METHOD SetPowerMode : BOOL
VAR_INST
	WriteReg	:	FB_MBWriteSingleReg;
	Value 		:	WORD 	:= 1;
	StartWrite	:	BOOL	:= FALSE;
	bCommBusy	:	BOOL;
	bComError	:	BOOL;
	errID		:	UDINT;
	TransmissionDone 	: 	f_trig;
	ComTrigger	:	Ton := (PT := TIME#200MS);
	ComRetryCounter	:	USINT	:= 0;
END_VAR	

VAR

END_VAR

Value := ePowerControl.Stay; //default command is: Do nothing
//it may also work if we just keep sending "poweron" if b_HVDC_Required is true. But this doesn't seem to be the way they intended.

IF Set.b_HVDC_Required AND (BMSGet.BattInfo.ui_BMS_PowerOnStatus = ePowerOnStatus.Off) THEN	//send poweron if system not already on
	Value := ePowerControl.PowerOn;
ELSIF (NOT Set.b_HVDC_Required) AND (BMSGet.BattInfo.ui_BMS_PowerOnStatus = ePowerOnStatus.On) THEN //send poweroff if system not already off
	Value := ePowerControl.PowerOff;
END_IF

//Write this register every second, regardless of change.
ComTrigger(in := NOT(ComTrigger.Q));

//IF BMSGet.BattInfo.ui_BMS_Status < 5 THEN
WriteReg(
	sIPAddr := Config.IP_BMS,
	nTCPPort := Config.MBPort_BMS,
	nUnitID := 255,//16#FF;
	nMBAddr := 897,
	nValue := Value,
	tTimeout := T#0S100MS,
	bExecute := ComTrigger.Q,
	bBusy => bCommBusy,
	bError => bComError,
	nErrId => errID,
);
//ELSE
//	SetPowerMode := TRUE;
//END_IF

	
TransmissionDone(CLK := bCommBusy);
	
//return true if tranmission succeeds
IF TransmissionDone.Q THEN
	IF NOT bComError THEN
		SetPowerMode := TRUE;
		ComRetryCounter := 0;
	ELSE
		COMretryCounter := COMretryCounter +1;
		IF COMRetryCounter > 5 THEN
			b_MBComErrorActive := TRUE;
		END_IF
	END_IF
END_IF
END_METHOD

ACTION SFCTipReset:
SFCTip := FALSE;
END_ACTION

END_FUNCTION_BLOCK

// ---- POUs/Objects/BMS/FB_BMS_IO.TcPOU
FUNCTION_BLOCK FB_BMS_IO

VAR_INPUT
	HWControl			:	st_BMS_IO;
END_VAR

VAR_OUTPUT
	BMSPowerControl			AT %Q* : st_BMS_IO;
END_VAR

VAR
	PowerUpDelay	:	TON := (PT := TIME#1s0ms);
END_VAR


BMSPowerControl.b_BMS_230V_Enable := HWControl.b_BMS_230V_Enable;
BMSPowerControl.b_BMS_24V_Enable	:= HWControl.b_BMS_24V_Enable;

END_FUNCTION_BLOCK

// ---- POUs/Objects/CoolingSystem/CoolingStack/FB_Heatpump.TcPOU
FUNCTION_BLOCK FB_Heatpump
VAR
	u_counter: UINT;
	InitSFC			:	FB_HeatPumpInit;
	OperationSFC	:	FB_HeatPumpOperation;
	
	//only written once at init.
	HeatPumpID		:	BYTE := 0;
END_VAR

VAR_STAT
	ui_Instancecounter : byte := 0;
END_VAR

VAR	
	MBMaster				: 	ModbusRtuMasterV2_KL6x22B;
	
	DataBuffer				:	ARRAY[0..50] OF WORD;
//	b_MBBusy				:	BOOL;
//	b_MBerr					:	BOOL;
//	ui_cbRead				:	UINT;
//	b_EnableTransmission	:	BOOL;
//	ModbusStartTrigger		:	R_Trig;
//	MBRetryCount			:	BYTE;
	
	
//	SendValue		:	WORD;
	
	OperatingPoint	:	st_OperatingPoint;
END_VAR

VAR_OUTPUT
	get			:	st_HeatpumpGet;
	MBCommBusy	:	BOOL := FALSE;
END_VAR

VAR_INPUT
	ACPowerStatus	:	BOOL;
	MBFree			:	BOOL;
END_VAR

//HeatpumpId is set once during first call
//var Stat InstanceCounter is shared between all functionblocks
IF HeatPumpId = 0 THEN
	ui_Instancecounter := ui_Instancecounter + 1;
	HeatPumpID := ui_Instancecounter ;
ELSE
	IF NOT ACPowerStatus THEN
		//Dont read all sensor data. Just monitor errors. We are not going to do anyting with the data anyway.
		InitSFC.SFCInit := TRUE;
		OperationSFC.SFCInit := TRUE;
		//OperationalSFC();
	ELSE
		InitSFC.SFCInit := FALSE;
		OperationSFC.SFCInit := FALSE;
	END_IF
END_IF

InitSFC(MBMaster := MBMaster, Get := Get, ACPowerSTatus := ACPowerStatus, HeatPumpID:=HeatPumpID);
OperationSFC(MBMaster := MBMaster, Get := Get, ACPowerSTatus := ACPowerStatus, HeatPumpID:=HeatPumpID,MBFree:=MBFree, OperatingPoint:=OperatingPoint, MBCommBusy=>MBCommbusy);

METHOD EMStop : BOOL
VAR_INPUT
END_VAR

get.HeatPumpState := eHeatpumpState.OFF;

EMstop := True;
END_METHOD

METHOD GetDiagnostics 
VAR_IN_OUT
	AddError		: ARRAY [*] OF FB_AddErrorST;
	a_ActiveEvents	: ARRAY [*] OF ST_ErrorStruct;
	w_Index			: WORD;
END_VAR

VAR_OUTPUT
	b_errorActive	: BOOL;
	b_warningActive	: BOOL;
END_VAR

VAR
	by_errCt	: BYTE;
	by_warnCt	: BYTE;
	w_ID		: WORD;
END_VAR
	(*Modbus comm fault*)	AddError[w_Index](
			in_b_ErrorTrig			:= Get.Events.b_CommError,
			out_ST_Error			:= a_ActiveEvents[w_Index],
			w_ID					:= 1 + w_ID,
			s_Message				:= 'Modbus communication error',
			e_sev					:= eSeverity.NormalShutdown,	
			in_b_AutoClear			:= FALSE,
			//in_e_ErrAckAccess		:= TRUE,
			);
		IF AddError[w_Index].b_out THEN by_errCt := by_errCt + 1; END_IF;
		w_Index := w_Index +1;
		
	(*Heatpump Compressor fault*)	AddError[w_Index](
			in_b_ErrorTrig			:= Get.Events.b_CompressorError,
			out_ST_Error			:= a_ActiveEvents[w_Index],
			w_ID					:= 2 + w_ID,
			s_Message				:= 'Heatpump Compressor fault',
			e_sev					:= eSeverity.NormalShutdown,	
			in_b_AutoClear			:= FALSE,
			//in_e_ErrAckAccess		:= TRUE,
			);
		IF AddError[w_Index].b_out THEN by_errCt := by_errCt + 1; END_IF;
		w_Index := w_Index +1;
	
	(*Heatpump Fan fault*)			AddError[w_Index](
			in_b_ErrorTrig			:= Get.Events.b_FanError,
			out_ST_Error			:= a_ActiveEvents[w_Index],
			w_ID					:= 3 + w_ID,
			s_Message				:= 'Heatpump Fan fault',
			e_sev					:= eSeverity.NormalShutdown,	
			in_b_AutoClear			:= FALSE,
			//in_e_ErrAckAccess		:= TRUE,
			);
		IF AddError[w_Index].b_out THEN by_errCt := by_errCt + 1; END_IF;
		w_Index := w_Index +1;
		
	(*HHeatpump Internal IO fault*)		AddError[w_Index](
			in_b_ErrorTrig			:= Get.Events.b_IOError ,
			out_ST_Error			:= a_ActiveEvents[w_Index],
			w_ID					:= 4 + w_ID,
			s_Message				:= 'Heatpump Internal IO fault',
			e_sev					:= eSeverity.NormalShutdown,	
			in_b_AutoClear			:= FALSE,
			//in_e_ErrAckAccess		:= TRUE,
			);
		IF AddError[w_Index].b_out THEN by_errCt := by_errCt + 1; END_IF;
		w_Index := w_Index +1;
		
	(*Heatpump pressure fault*)		AddError[w_Index](
			in_b_ErrorTrig			:= Get.Events.b_PressureError,
			out_ST_Error			:= a_ActiveEvents[w_Index],
			w_ID					:= 5 + w_ID,
			s_Message				:= 'Heatpump pressure fault',
			e_sev					:= eSeverity.NormalShutdown,	
			in_b_AutoClear			:= FALSE,
			//in_e_ErrAckAccess		:= TRUE,
			);
		IF AddError[w_Index].b_out THEN by_errCt := by_errCt + 1; END_IF;
		w_Index := w_Index +1;
		
	(*Heatpump Probe fault*)		AddError[w_Index](
			in_b_ErrorTrig			:= Get.Events.b_ProbeError,
			out_ST_Error			:= a_ActiveEvents[w_Index],
			w_ID					:= 6 + w_ID,
			s_Message				:= 'Heatpump Probe fault',
			e_sev					:= eSeverity.NormalShutdown,	
			in_b_AutoClear			:= FALSE,
			//in_e_ErrAckAccess		:= TRUE,
			);
		IF AddError[w_Index].b_out THEN by_errCt := by_errCt + 1; END_IF;
		w_Index := w_Index +1;	

	(*Heatpump Pump fault*)			AddError[w_Index](
			in_b_ErrorTrig			:= Get.Events.b_PumpError,
			out_ST_Error			:= a_ActiveEvents[w_Index],
			w_ID					:= 7 + w_ID,
			s_Message				:= 'Heatpump Pump fault',
			e_sev					:= eSeverity.NormalShutdown,	
			in_b_AutoClear			:= FALSE,
			//in_e_ErrAckAccess		:= TRUE,
			);
		IF AddError[w_Index].b_out THEN by_errCt := by_errCt + 1; END_IF;
		w_Index := w_Index +1;	

	(*Heatpump valve fault*)			AddError[w_Index](
			in_b_ErrorTrig			:= Get.Events.b_ValveError,
			out_ST_Error			:= a_ActiveEvents[w_Index],
			w_ID					:= 8 + w_ID,
			s_Message				:= 'Heatpump Valve fault',
			e_sev					:= eSeverity.NormalShutdown,	
			in_b_AutoClear			:= FALSE,
			//in_e_ErrAckAccess		:= TRUE,
			);
		IF AddError[w_Index].b_out THEN by_errCt := by_errCt + 1; END_IF;
		w_Index := w_Index +1;	

	(*Heatpump Water temperature error*)			AddError[w_Index](
			in_b_ErrorTrig			:= Get.Events.b_WaterTempError,
			out_ST_Error			:= a_ActiveEvents[w_Index],
			w_ID					:= 9 + w_ID,
			s_Message				:= 'Heatpump Water temperature error',
			e_sev					:= eSeverity.NormalShutdown,	
			in_b_AutoClear			:= FALSE,
			//in_e_ErrAckAccess		:= TRUE,
			);
		IF AddError[w_Index].b_out THEN by_errCt := by_errCt + 1; END_IF;
		w_Index := w_Index +1;	

(*Heatpump Comm warning*)			AddError[w_Index](
			in_b_ErrorTrig			:= Get.Events.b_commwarning,
			out_ST_Error			:= a_ActiveEvents[w_Index],
			w_ID					:= 10 + w_ID,
			s_Message				:= 'Heatpump communication warning',
			e_sev					:= eSeverity.Info,	
			in_b_AutoClear			:= TRUE,
			//in_e_ErrAckAccess		:= TRUE,
			);
		
		//for initial use, get notice if 1 packet fails. Clear immediately after datalogger run
		get.Events.b_CommWarning := FALSE;
END_METHOD

METHOD Reset : BOOL
VAR_INPUT
END_VAR
//until restarting the heatpump we don't know if errors are gone. So clear them for now.

get.Events.b_CommError := FALSE;
get.Events.b_CompressorError := FALSE;
get.Events.b_FanError := FALSE;
get.Events.b_IOError := FALSE;
get.Events.b_PressureError := FALSE;
get.Events.b_ProbeError := FALSE;
get.Events.b_PumpError := FALSE;
get.Events.b_ValveError := FALSE;
get.Events.b_WaterTempError := FALSE;

Reset := True;
END_METHOD

METHOD WriteSetpoint : BOOL
VAR_INPUT
	OperatingMode	:	eHeatpumpMode;
	SetPoint		: 	REAL;
END_VAR


OperatingPoint.OperatingMode := OperatingMode;
OperatingPoint.Setpoint := SetPoint;
END_METHOD

END_FUNCTION_BLOCK

// ---- POUs/Objects/CoolingSystem/CoolingStack/SFC/FB_HeatpumpInit.TcPOU
FUNCTION_BLOCK FB_HeatpumpInit
VAR_IN_OUT
	MBMaster		:	ModbusRtuMasterV2_KL6x22B;
	Get				:	ST_HeatpumpGet;
END_VAR

VAR_INPUT
	ACPowerStatus	:	BOOL;
	HeatPumpID		:	BYTE;
	SFCInit			:	BOOL;
END_VAR
		
VAR
	TransmissionDone		:	BOOL;
	DataBuffer				:	ARRAY[0..50] OF WORD;
	b_MBBusy				:	BOOL;
	b_MBerr					:	BOOL;
	ui_cbRead				:	UINT;
	b_EnableTransmission	:	BOOL;
	ModbusRetryTimer		:	TON := (PT := TIME#250MS);
	ModbusStartTrigger		:	R_Trig;
	TransmissionDoneTrigger	:	F_Trig;
	MBRetryCount			:	BYTE;
	u_Counter				:	uint;
	
	SendValue		:	WORD;
	
	w_errid: Tc2_ModbusRTU.MODBUS_ERRORS;
	ResetRetryTimer: BOOL;
END_VAR
VAR_OUTPUT
END_VAR
VAR
END_VAR

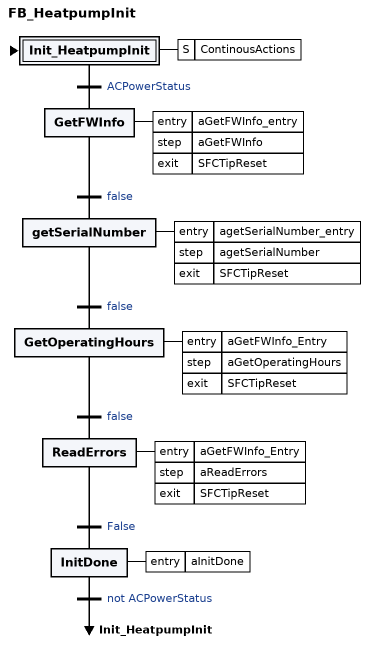
INITIAL_STEP Init_HeatpumpInit:
    ContinousActions(S);
END_STEP
TRANSITION FROM Init_HeatpumpInit TO GetFWInfo
    := ACPowerStatus;
END_TRANSITION
STEP GetFWInfo:
    aGetFWInfo_entry(P1);  // entry action
    aGetFWInfo(N);  // step action
    SFCTipReset(P0);  // exit action
END_STEP
TRANSITION FROM GetFWInfo TO getSerialNumber
    := false;
END_TRANSITION
STEP getSerialNumber:
    agetSerialNumber_entry(P1);  // entry action
    agetSerialNumber(N);  // step action
    SFCTipReset(P0);  // exit action
END_STEP
TRANSITION FROM getSerialNumber TO GetOperatingHours
    := false;
END_TRANSITION
STEP GetOperatingHours:
    aGetFWInfo_Entry(P1);  // entry action
    aGetOperatingHours(N);  // step action
    SFCTipReset(P0);  // exit action
END_STEP
TRANSITION FROM GetOperatingHours TO ReadErrors
    := false;
END_TRANSITION
STEP ReadErrors:
    aGetFWInfo_Entry(P1);  // entry action
    aReadErrors(N);  // step action
    SFCTipReset(P0);  // exit action
END_STEP
TRANSITION FROM ReadErrors TO InitDone
    := False;
END_TRANSITION
STEP InitDone:
    aInitDone(P1);  // entry action
END_STEP
TRANSITION FROM InitDone TO Init_HeatpumpInit
    := not ACPowerStatus;
END_TRANSITION

ACTION aGetFWInfo:

//ModbusStartTrigger(clk := b_EnableTransmission);

IF NOT b_enableTransmission THEN
	b_enableTransmission := TRUE;
END_IF

MBMaster.ReadRegs(	UnitID 		:= 	HeatPumpID,
					Quantity 	:= 	4,
					MBAddr		:=	1,
					cbLength 	:= 	64,
					pMemoryAddr	:=	ADR(DataBuffer),
					Execute		:=	ModbusStartTrigger.Q,
					Timeout		:=	T#250MS,		
					Busy		=>	b_MBBusy,
					Error 		=>	b_MBerr,
					cbRead 		=>	ui_cbRead,
					ErrorId		=>	w_errid
					);


TransmissionDoneTrigger(clk := b_MBBusy);

IF TransmissionDoneTrigger.q THEN
	IF NOT b_MBerr THEN
		get.HeatpumpData.i_FW_Version 		:= 	WORD_TO_INT(DataBuffer[0]);
		get.HeatpumpData.i_FW_release 		:= 	WORD_TO_INT(DataBuffer[1]);
		get.HeatpumpData.w_FW_Subrelease 	:= 	DataBuffer[2];
		get.HeatpumpData.w_FW_creationDate	:=	DataBuffer[3];
			
		TransmissionDone := TRUE;
		//done, preset for next step
		//b_EnableTransmission := FALSE;
		//ModbusStartTrigger(clk := b_EnableTransmission);
		MBRetryCount := 0;
		//ResetRetryTimer := TRUE;
		
		sfctip := TRUE;
	ELSE
		MBRetryCount := MBRetryCount + 1;
		b_EnableTransmission	:= FALSE;
		
		//if heatpump is still unreachable after 1 minute, something failed during poweron
		IF MBRetryCount > 240 THEN
			get.HeatPumpState := eHeatpumpState.ERROR;
			get.Events.b_CommError := TRUE;
		END_IF
	END_IF
END_IF



(*
IF b_EnableTransmission AND NOT b_MBBusy[0] THEN
	IF NOT b_MBerr[0] THEN
			//transmission done, process data
			get.HeatpumpData.i_FW_Version 		:= 	WORD_TO_INT(DataBuffer[0]);
			get.HeatpumpData.i_FW_release 		:= 	WORD_TO_INT(DataBuffer[1]);
			get.HeatpumpData.w_FW_Subrelease 	:= 	DataBuffer[2];
			get.HeatpumpData.w_FW_creationDate	:=	DataBuffer[3];
			
			TransmissionDone := TRUE;
			//done, preset for next step
			//b_EnableTransmission := FALSE;
			//ModbusStartTrigger(clk := b_EnableTransmission);
			MBRetryCount := 0;
	
			//sfctip := TRUE;
		ELSE
			MBRetryCount := MBRetryCount + 1;
			
			//add comm error functionality later
			IF MBRetryCount < 10 THEN
				//retry
				b_EnableTransmission	:= FALSE;
			ELSE
				//do something else
				b_EnableTransmission	:= FALSE;
			END_IF
		END_IF
	END_IF


IF TransmissionDone THEN
	sfctip := TRUE;
END_IF


IF NOT b_MBBusy[0] THEN
	IF NOT b_MBerr[0] THEN
		//transmission done, process data
		get.HeatpumpData.i_FW_Version 		:= 	WORD_TO_INT(DataBuffer[0]);
		get.HeatpumpData.i_FW_release 		:= 	WORD_TO_INT(DataBuffer[1]);
		get.HeatpumpData.w_FW_Subrelease 	:= 	DataBuffer[2];
		get.HeatpumpData.w_FW_creationDate	:=	DataBuffer[3];
		
		//done, preset for next step
		b_EnableTransmission := FALSE;
		ModbusStartTrigger(clk := b_EnableTransmission);
		MBRetryCount := 0;

		sfctip := TRUE;
	ELSE
		MBRetryCount := MBRetryCount + 1;
		
		//add comm error functionality later
		IF MBRetryCount < 10 THEN
			//retry
			b_EnableTransmission	:= FALSE;
		ELSE
			//do something else
			b_EnableTransmission	:= FALSE;
		END_IF
	END_IF
END_IF
*)
END_ACTION

ACTION aGetFWInfo_entry:
//ResetRetryTimer := TRUE;
//TransmissionDone := False;

get.HeatPumpState := eHeatpumpState.Initializing;
END_ACTION

ACTION aGetOperatingHours:


MBMaster.ReadRegs(	UnitID 		:= 	HeatPumpID,
					Quantity 	:= 	1,
					MBAddr		:=	305,
					cbLength 	:= 	1*2,
					pMemoryAddr	:=	ADR(DataBuffer),
					Execute		:=	ModbusStartTrigger.Q,
					Timeout		:=	T#250MS,		
					Busy		=>	b_MBBusy,
					Error 		=>	b_MBerr,
					cbRead 		=>	ui_cbRead,
					ErrorId		=>	w_errid
					);

TransmissionDoneTrigger(clk := b_MBBusy);

IF TransmissionDoneTrigger.q THEN
	IF NOT b_MBerr THEN
		//transmission done, process data
		
		//just use comp 1 for now. See if the others are even used
		//i think it will be a dual word value. But check later
		get.HeatpumpData.i_OperatingHours := WORD_TO_INT(DataBuffer[0]);
		
		//done, preset for next step
		b_EnableTransmission := FALSE;
//		ModbusStartTrigger(clk := b_EnableTransmission);
		MBRetryCount := 0;
		sfctip := TRUE;
	ELSE
		MBRetryCount := MBRetryCount + 1;
		b_EnableTransmission	:= FALSE;
		
		//if comm fails 5 times in a row. system is unusable
		IF MBRetryCount > 5 THEN
			get.HeatPumpState := eHeatpumpState.ERROR;
			get.Events.b_CommError := TRUE;
		END_IF
	END_IF
END_IF
END_ACTION

ACTION agetSerialNumber:



IF NOT b_enableTransmission THEN
	b_enableTransmission := TRUE;
END_IF


MBMaster.ReadRegs(	UnitID 		:= 	HeatPumpID,
					Quantity 	:= 	18,
					MBAddr		:=	80,
					cbLength 	:= 	32*2,
					pMemoryAddr	:=	ADR(DataBuffer),
					Execute		:=	ModbusStartTrigger.Q,
					Timeout		:=	T#250MS,		
					Busy		=>	b_MBBusy,
					Error 		=>	b_MBerr,
					cbRead 		=>	ui_cbRead,
					ErrorId		=>	w_errid
					);

TransmissionDoneTrigger(clk := b_MBBusy);

IF TransmissionDoneTrigger.q THEN
	IF NOT b_MBerr THEN
		FOR u_counter:=0 TO 17 BY 1 DO
			get.HeatpumpData.w_Serialnumber[u_counter]	:= 	DataBuffer[u_counter];
		END_FOR
			
		TransmissionDone := TRUE;
		//done, preset for next step
		//b_EnableTransmission := FALSE;
		//ModbusStartTrigger(clk := b_EnableTransmission);
		MBRetryCount := 0;
	
		sfctip := TRUE;
	ELSE
		MBRetryCount := MBRetryCount + 1;
		b_EnableTransmission	:= FALSE;
		
		//if comm fails 5 times in a row. system is unusable
		IF MBRetryCount > 5 THEN
			get.HeatPumpState := eHeatpumpState.ERROR;
			get.Events.b_CommError := TRUE;
		END_IF
	END_IF
END_IF

(*
IF b_EnableTransmission AND NOT b_MBBusy[2] THEN
	IF NOT b_MBerr[2] THEN
		//transmission done, process data

		
		//maybe try to put get struct directly in MBREAD pMemoryAddr later
		FOR u_counter:=0 TO 8 BY 1 DO
			get.HeatpumpData.w_Serialnumber[u_counter]	:= 	DataBuffer[u_counter];
		END_FOR
			
			TransmissionDone := TRUE;
			//done, preset for next step
			//b_EnableTransmission := FALSE;
			//ModbusStartTrigger(clk := b_EnableTransmission);
			MBRetryCount := 0;
	
			//sfctip := TRUE;
		ELSE
			MBRetryCount := MBRetryCount + 1;
			
			//add comm error functionality later
			IF MBRetryCount < 10 THEN
				//retry
				b_EnableTransmission	:= FALSE;
			ELSE
				//do something else
				b_EnableTransmission	:= FALSE;
			END_IF
		END_IF
	END_IF


IF TransmissionDone THEN
	sfctip := TRUE;
END_IF
		
				
IF NOT b_MBBusy[2] THEN
	IF NOT b_MBerr[2] THEN
		//transmission done, process data
		
		//maybe try to put get struct directly in MBREAD pMemoryAddr later
		FOR u_counter:=0 TO 8 BY 1 DO
			get.HeatpumpData.w_Serialnumber[u_counter]	:= 	DataBuffer[u_counter];
		END_FOR
		
		//done, preset for next step
		b_EnableTransmission := FALSE;
		ModbusStartTrigger(clk := b_EnableTransmission);
		MBRetryCount := 0;
		sfctip := TRUE;
	ELSE
		MBRetryCount := MBRetryCount + 1;
		
		//add comm error functionality later
		IF MBRetryCount < 10 THEN
			//retry
			b_EnableTransmission	:= FALSE;
		ELSE
			//do something else
			b_EnableTransmission	:= FALSE;
		END_IF
	END_IF
END_IF
*)
END_ACTION

ACTION agetSerialNumber_entry:
//SFCTip := FALSE;
//TransmissionDone := False;
END_ACTION

ACTION aInitDone:
SFCTip := FALSE;
IF get.HeatPumpState = eHeatPumpState.Initializing THEN
	get.HeatPumpState := eHeatPumpState.Standby;
end_if
END_ACTION

ACTION aReadErrors:
//SFCTip := FALSE;
//b_EnableTransmission	:= TRUE;
//ModbusStartTrigger(clk := b_EnableTransmission);

MBMaster.ReadRegs(	UnitID 		:= 	HeatPumpID,
					Quantity 	:= 	7,
					MBAddr		:=	950,
					cbLength 	:= 	7*2,
					pMemoryAddr	:=	ADR(DataBuffer),
					Execute		:=	ModbusStartTrigger.Q,
					Timeout		:=	T#500MS,		
					Busy		=>	b_MBBusy,
					Error 		=>	b_MBerr,
					cbRead 		=>	ui_cbRead,
					ErrorId		=>	w_errid
					);

TransmissionDoneTrigger(clk := b_MBBusy);

IF TransmissionDoneTrigger.q THEN
	IF NOT b_MBerr THEN
		//transmission done, process data
		
		ParseHeatPumpErrors(	w_Alarms1 := DataBuffer[0],
								w_Alarms2 := DataBuffer[1],
								w_Alarms3 := DataBuffer[2],
								w_Alarms4 := DataBuffer[3],
								w_Alarms5 := DataBuffer[4],
								w_Alarms6 := DataBuffer[5],
								w_Alarms7 := DataBuffer[6],
								Get := Get				
							);
		
		//done, preset for next step
		b_EnableTransmission := FALSE;
//		ModbusStartTrigger(clk := b_EnableTransmission);
		MBRetryCount := 0;
		sfctip := TRUE;
	ELSE
		MBRetryCount := MBRetryCount + 1;
		b_EnableTransmission	:= FALSE;
		
		//if comm fails 5 times in a row. system is unusable
		IF MBRetryCount > 5 THEN
			get.HeatPumpState := eHeatpumpState.ERROR;
			get.Events.b_CommError := TRUE;
		END_IF
	END_IF
END_IF
END_ACTION

ACTION ContinousActions:
//sfctip := False;
ModbusRetryTimer(in:= NOT (ModbusRetryTimer.Q OR ResetRetryTimer));
ModbusStartTrigger(clk := ModbusRetryTimer.Q);

//for initial use, get notice if 1 packet fails
IF MBRetryCount > 1 THEN
	get.Events.b_CommWarning := TRUE;
END_IF

//ResetRetryTimer := FALSE;
END_ACTION

METHOD ParseHeatPumpErrors : BOOL
VAR_INPUT
	w_Alarms1	:	WORD;
	w_Alarms2	:	WORD;
	w_Alarms3	:	WORD;
	w_Alarms4	:	WORD;
	w_Alarms5	:	WORD;
	w_Alarms6	:	WORD;
	w_Alarms7	:	WORD;
END_VAR		
VAR_IN_OUT
	get	:	ST_HeatpumpGet;	
END_VAR

get.events.b_ProbeError		:=	WORD_TO_BOOL(w_Alarms3) OR WORD_TO_BOOL(w_Alarms4) OR w_Alarms5.0;

get.events.b_PressureError		:=	w_Alarms1.0 OR	//E001: High Pressure
									w_Alarms1.1 OR //E002: Low Pressure
									w_Alarms2.3;	//E020: Inverted Pressure Transducers


get.events.b_CompressorError	:=	w_Alarms1.2 OR //E003: Compressor overheated
									w_Alarms1.7 OR //E008: Compressor underspeed
									w_Alarms1.8 OR	//E009: High disch temp
									w_Alarms1.12 OR //E013: Comp2 Overheated
									w_Alarms2.2 OR	//E019: CP2 High disch temp
									w_Alarms2.6 OR	//E023: Comp3 Overheated
									w_Alarms5.1 OR //'E801: Link Inverter1',
									w_Alarms5.2 OR //'E802: Link Inverter2',
									w_Alarms5.3 OR //'E803: Link Inverter3',
									w_Alarms5.4 OR //'E851: HWfault Inverter1',
									w_Alarms5.5 OR //'E852: HWfault Inverter2',
									w_Alarms5.6 OR //'E853: HWfault Inverter3',
									w_Alarms5.7 OR //'E861: OverCurrent Inv1',
									w_Alarms5.8 OR //'E862: OverCurrent Inv2',
									w_Alarms5.9 OR //'E863: OverCurrent Inv3',
									w_Alarms5.10 OR //'E871: High Temp Inv1',
									w_Alarms5.11 OR //'E872: High Temp Inv2',
									w_Alarms5.12 OR //'E873: High Temp Inv3',
									w_Alarms5.13 OR //'E881: Bad Voltage Inv1',
									w_Alarms5.14 OR //'E882: Bad Voltage Inv2',
									w_Alarms5.15 OR //'E883: Bad Voltage Inv3',
									w_Alarms6.0 OR //E891: Phase Seq Inv1',
									w_Alarms6.1 OR //'E892: Phase Seq Inv2',
									w_Alarms6.2 OR //'E893: Phase Seq Inv3',
									w_Alarms6.3 OR //'E901: Model err Inv1',
									w_Alarms6.4 OR //'E902: Model err Inv2',
									w_Alarms6.5 OR //'E903: Model err Inv3',
									w_Alarms6.6 OR //'E911: Ovl error Inv1',
									w_Alarms6.7 OR //'E9112: Ovl error Inv2',
									w_Alarms6.8 OR //'E913: Ovl error Inv3',
									w_Alarms6.9 OR //'E921: Overc PFC Inv1',
									w_Alarms6.10 OR //'E922: Overc PFC Inv2',
									w_Alarms6.11 OR //'E923: Overc PFC Inv3',
									w_Alarms6.12 OR //'E931: Int Com ERR Inv1',
									w_Alarms6.13 OR //'E932: Int Com ERR Inv2',
									w_Alarms6.14 OR //'E933: Int Com ERR Inv3',
									w_Alarms6.15 OR //'E941: Fault PFC Inv1',
									w_Alarms7.0 OR //E942: Fault PFC Inv2
									w_Alarms7.1 OR //'E943: Fault PFC Inv3',
									w_Alarms7.2 OR //'E951: Probe error Inv1',
									w_Alarms7.3 OR //'E952: Probe error Inv2',
									w_Alarms7.4 OR //'E953: Probe error Inv3',
									w_Alarms7.5 OR //'E961: Abnormal Cond Inv1',
									w_Alarms7.6 OR //'E962: Abnormal Cond Inv2',
									w_Alarms7.7 OR //'E963: Abnormal Cond Inv3',
									w_Alarms7.8 OR //'E971: Inv1 Eeprom Error',
									w_Alarms7.9 OR //'E972: Inv2 Eeprom Error',
									w_Alarms7.10 OR //'E973: Inv3 Eeprom Error',
									w_Alarms7.11;	//E029: CP3 High disch temp

get.events.b_ValveError		:=		w_Alarms2.11; //E041: Incongruent temps;


get.events.b_FanError			:=	w_Alarms1.2 OR //E004: Fan Overheated	
									w_Alarms1.13 OR //E014: Fan2 Overheated 
									w_Alarms2.7;	//E024: Fan3 Overheated					

get.events.b_PumpError			:=	w_Alarms1.5 OR	 	//E006: Lack of flow
									w_Alarms1.15 OR 	//E016: Pump Overheated
									w_Alarms2.9;		//E026: Pump2 Overheated

get.events.b_WaterTempError		:=	w_Alarms2.1 OR	//E018: OverTemperature
									w_Alarms1.4;	//E005: Frost

get.events.b_IOError			:=	w_Alarms2.14 OR 	//E101: IOMod1 Disconnected
									w_Alarms2.15; 		//E102: IOMod2 Disconnected
END_METHOD

ACTION SFCTipReset:
SFCTip := FALSE;
ResetRetryTimer := FALSE;
END_ACTION

END_FUNCTION_BLOCK

// ---- POUs/Objects/CoolingSystem/CoolingStack/SFC/FB_HeatpumpOperation.TcPOU
FUNCTION_BLOCK FB_HeatpumpOperation
VAR_IN_OUT
	MBMaster		:	ModbusRtuMasterV2_KL6x22B;
	Get				:	ST_HeatpumpGet;
END_VAR

VAR_INPUT
	ACPowerStatus	:	BOOL;
	HeatPumpID		:	BYTE;
	MBFree			:	BOOL;
	OperatingPoint	:	st_OperatingPoint;
	SFCInit			:	BOOL;
END_VAR
		
VAR
	DataBuffer				:	ARRAY[0..50] OF WORD;
	b_MBBusy				:	BOOL;
	b_MBerr					:	BOOL;
	ui_cbRead				:	UINT;
	b_EnableTransmission	:	BOOL;
	ModbusStartTrigger		:	R_Trig;
	MBRetryCount			:	BYTE;
	ModbusRetryTimer		:	TON := (PT := TIME#250MS);
	ResetRetryTimer			:	Bool;
	SendValue		:	WORD;
	TransmissionDoneTrigger	:	F_Trig;
	
	ReadSetpointHeating		:	REAL;
	ReadSetpointCooling		:	REAL;
	ReadCoolingMode			:	WORD;
	Writeregstatus			:	WORD;
END_VAR

VAR_OUTPUT
	MBCommBusy				:	Bool;
END_VAR

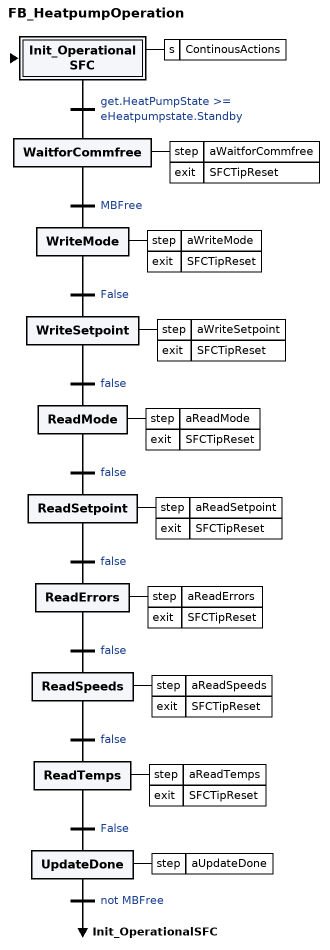
INITIAL_STEP Init_OperationalSFC:
    ContinousActions(s);
END_STEP
TRANSITION FROM Init_OperationalSFC TO WaitforCommfree
    := get.HeatPumpState >= eHeatpumpstate.Standby;
END_TRANSITION
STEP WaitforCommfree:
    aWaitforCommfree(N);  // step action
    SFCTipReset(P0);  // exit action
END_STEP
TRANSITION FROM WaitforCommfree TO WriteMode
    := MBFree;
END_TRANSITION
STEP WriteMode:
    aWriteMode(N);  // step action
    SFCTipReset(P0);  // exit action
END_STEP
TRANSITION FROM WriteMode TO WriteSetpoint
    := False;
END_TRANSITION
STEP WriteSetpoint:
    aWriteSetpoint(N);  // step action
    SFCTipReset(P0);  // exit action
END_STEP
TRANSITION FROM WriteSetpoint TO ReadMode
    := false;
END_TRANSITION
STEP ReadMode:
    aReadMode(N);  // step action
    SFCTipReset(P0);  // exit action
END_STEP
TRANSITION FROM ReadMode TO ReadSetpoint
    := false;
END_TRANSITION
STEP ReadSetpoint:
    aReadSetpoint(N);  // step action
    SFCTipReset(P0);  // exit action
END_STEP
TRANSITION FROM ReadSetpoint TO ReadErrors
    := false;
END_TRANSITION
STEP ReadErrors:
    aReadErrors(N);  // step action
    SFCTipReset(P0);  // exit action
END_STEP
TRANSITION FROM ReadErrors TO ReadSpeeds
    := false;
END_TRANSITION
STEP ReadSpeeds:
    aReadSpeeds(N);  // step action
    SFCTipReset(P0);  // exit action
END_STEP
TRANSITION FROM ReadSpeeds TO ReadTemps
    := false;
END_TRANSITION
STEP ReadTemps:
    aReadTemps(N);  // step action
    SFCTipReset(P0);  // exit action
END_STEP
TRANSITION FROM ReadTemps TO UpdateDone
    := False;
END_TRANSITION
STEP UpdateDone:
    aUpdateDone(N);  // step action
END_STEP
TRANSITION FROM UpdateDone TO Init_OperationalSFC
    := not MBFree;
END_TRANSITION

ACTION aReadErrors:

MBMaster.ReadRegs(	UnitID 		:= 	HeatPumpID,
					Quantity 	:= 	7,
					MBAddr		:=	950,
					cbLength 	:= 	7*2,
					pMemoryAddr	:=	ADR(DataBuffer),
					Execute		:=	ModbusStartTrigger.Q,
					Timeout		:=	T#250MS,		
					Busy		=>	b_MBBusy,
					Error 		=>	b_MBerr,
					cbRead 		=>	ui_cbRead
					);

TransmissionDoneTrigger(clk := b_MBBusy);

IF TransmissionDoneTrigger.q THEN
	IF NOT b_MBerr THEN
		
		ParseHeatPumpErrors(	w_Alarms1 := DataBuffer[0],
								w_Alarms2 := DataBuffer[1],
								w_Alarms3 := DataBuffer[2],
								w_Alarms4 := DataBuffer[3],
								w_Alarms5 := DataBuffer[4],
								w_Alarms6 := DataBuffer[5],
								w_Alarms7 := DataBuffer[6],
								Get := Get			
							);
		
		//done, preset for next step
		
		MBRetryCount := 0;
		sfctip := TRUE;
	ELSE
		MBRetryCount := MBRetryCount + 1;
		b_EnableTransmission	:= FALSE;
				
		//if comm fails 5 times in a row. system is unusable
		IF MBRetryCount > 5 THEN
			get.HeatPumpState := eHeatpumpState.ERROR;
			get.Events.b_CommError := TRUE;
		END_IF
	END_IF
END_IF
END_ACTION

ACTION aReadMode:

MBMaster.ReadRegs(	UnitID 		:= 	HeatPumpID,
					Quantity 	:= 	1,
					MBAddr		:=	200,
					cbLength 	:= 	10,
					pMemoryAddr	:=	ADR(DataBuffer),
					Execute		:=	ModbusStartTrigger.Q,
					Timeout		:=	T#250MS,		
					Busy		=>	b_MBBusy,
					Error 		=>	b_MBerr,
					cbRead 		=>	ui_cbRead
					);

TransmissionDoneTrigger(clk := b_MBBusy);

IF TransmissionDoneTrigger.q THEN
	IF NOT b_MBerr THEN
	
		//transmission done, process data
		CASE DataBuffer[0] OF
			0:	get.HeatPumpState := eHeatpumpState.Standby;
			1:	get.HeatPumpState := eHeatpumpState.Active_Cooling;
			2:	get.HeatPumpState := eHeatpumpState.Active_Heating;
		END_CASE
		
		//done, preset for next step
		b_EnableTransmission := FALSE;
		ModbusStartTrigger(clk := b_EnableTransmission);
		MBRetryCount := 0;
		sfctip := TRUE;
	ELSE
		MBRetryCount := MBRetryCount + 1;
		b_EnableTransmission	:= FALSE;
		
		//if comm fails 5 times in a row. system is unusable
		IF MBRetryCount > 5 THEN
			get.HeatPumpState := eHeatpumpState.ERROR;
			get.Events.b_CommError := TRUE;
		END_IF
	END_IF
END_IF
END_ACTION

ACTION aReadSetpoint:

//r_FanSpeedPCT			:	REAL;		//7000
//r_PumpSpeedPCT		:	REAL;		//7001

MBMaster.ReadRegs(	UnitID 		:= 	HeatPumpID,
					Quantity 	:= 	2,
					MBAddr		:=	7203,
					cbLength 	:= 	10,
					pMemoryAddr	:=	ADR(DataBuffer),
					Execute		:=	ModbusStartTrigger.Q,
					Timeout		:=	T#250MS,		
					Busy		=>	b_MBBusy,
					Error 		=>	b_MBerr,
					cbRead 		=>	ui_cbRead
					);

TransmissionDoneTrigger(clk := b_MBBusy);

IF TransmissionDoneTrigger.q THEN
	IF NOT b_MBerr THEN
	
		//transmission done, process data
		get.HeatpumpData.r_SetpointHeating	:=	DataBuffer[1]/10;
		get.HeatpumpData.r_SetpointCooling	:=	DataBuffer[0]/10;
			
		//done, preset for next step
		b_EnableTransmission := FALSE;
		ModbusStartTrigger(clk := b_EnableTransmission);
		MBRetryCount := 0;
		sfctip := TRUE;
	ELSE
		MBRetryCount := MBRetryCount + 1;
		b_EnableTransmission	:= FALSE;
		
		//if comm fails 5 times in a row. system is unusable
		IF MBRetryCount > 5 THEN
			get.HeatPumpState := eHeatpumpState.ERROR;
			get.Events.b_CommError := TRUE;
		END_IF
	END_IF
END_IF
END_ACTION

ACTION aReadSpeeds:

//r_FanSpeedPCT			:	REAL;		//7000
//r_PumpSpeedPCT		:	REAL;		//7001

MBMaster.ReadRegs(	UnitID 		:= 	HeatPumpID,
					Quantity 	:= 	2,
					MBAddr		:=	7000,
					cbLength 	:= 	4,
					pMemoryAddr	:=	ADR(DataBuffer),
					Execute		:=	ModbusStartTrigger.Q,
					Timeout		:=	T#250MS,		
					Busy		=>	b_MBBusy,
					Error 		=>	b_MBerr,
					cbRead 		=>	ui_cbRead
					);

TransmissionDoneTrigger(clk := b_MBBusy);

IF TransmissionDoneTrigger.q THEN
	IF NOT b_MBerr THEN
		
		//transmission done, process data
		get.HeatpumpData.r_FanSpeedPCT		:=	WORD_TO_REAL(DataBuffer[0])/10;
		get.HeatpumpData.r_PumpSpeedPCT		:= 	WORD_TO_REAL(DataBuffer[1])/10;
		
		//done, preset for next step
		b_EnableTransmission := FALSE;
		ModbusStartTrigger(clk := b_EnableTransmission);
		MBRetryCount := 0;
		sfctip := TRUE;
	ELSE
		MBRetryCount := MBRetryCount + 1;
		b_EnableTransmission	:= FALSE;
		
		//if comm fails 5 times in a row. system is unusable
		IF MBRetryCount > 5 THEN
			get.HeatPumpState := eHeatpumpState.ERROR;
			get.Events.b_CommError := TRUE;
		END_IF
	END_IF
END_IF
END_ACTION

ACTION aReadTemps:

(*
r_InletWaterTemp	:	REAL;		//400
r_OutletWaterTemp	:	REAL;		//401
r_HighPressure		:	REAL;		//406
r_LowPressure		:	REAL;		//414
r_CompInputTemp		:	REAL;		//422
r_OutdoorTemp		:	REAL;		//428
r_CompOutputTemp	:	REAL;		//433-435
ui_WaterFlowRate		:	uINT;		//444
*)

MBMaster.ReadRegs(	UnitID 		:= 	HeatPumpID,
					Quantity 	:= 	45,
					MBAddr		:=	400,
					cbLength 	:= 	90,
					pMemoryAddr	:=	ADR(DataBuffer),
					Execute		:=	ModbusStartTrigger.Q,
					Timeout		:=	T#250MS,		
					Busy		=>	b_MBBusy,
					Error 		=>	b_MBerr,
					cbRead 		=>	ui_cbRead
					);

TransmissionDoneTrigger(clk := b_MBBusy);

IF TransmissionDoneTrigger.q THEN
	IF NOT b_MBerr THEN
		
		//transmission done, process data
		get.HeatpumpData.r_InletWaterTemp		:=	WORD_TO_REAL(DataBuffer[0])/10;
		get.HeatpumpData.r_OutletWaterTemp		:= 	WORD_TO_REAL(DataBuffer[1])/10;
		get.HeatpumpData.r_HighPressure			:=	WORD_TO_REAL(DataBuffer[6])/100;
		get.HeatpumpData.r_LowPressure			:= 	WORD_TO_REAL(DataBuffer[14])/100;
		get.HeatpumpData.r_CompInputTemp		:=	WORD_TO_REAL(DataBuffer[22])/10;
		get.HeatpumpData.r_OutdoorTemp			:= 	WORD_TO_REAL(DataBuffer[28])/10;
		get.HeatpumpData.r_CompOutputTemp		:=	WORD_TO_REAL(DataBuffer[33])/10;	//comp dischyarge 1 for now
		get.HeatpumpData.ui_WaterFlowRate			:= 	DataBuffer[44];
		
		//done, preset for next step
		b_EnableTransmission := FALSE;
		ModbusStartTrigger(clk := b_EnableTransmission);
		MBRetryCount := 0;
		sfctip := TRUE;
	ELSE
		MBRetryCount := MBRetryCount + 1;
		b_EnableTransmission	:= FALSE;
		
		//if comm fails 5 times in a row. system is unusable
		IF MBRetryCount > 5 THEN
			get.HeatPumpState := eHeatpumpState.ERROR;
			get.Events.b_CommError := TRUE;
		END_IF
	END_IF
END_IF
END_ACTION

ACTION aUpdateDone:
SFCTip := FALSE;
MBCommBusy := False;
END_ACTION

ACTION aWaitforCommfree:
//SFCTip := FALSE;
//b_EnableTransmission	:= FALSE;
//ModbusStartTrigger(clk := b_EnableTransmission);
END_ACTION

ACTION aWriteMode:
//SFCTip := FALSE;


//b_EnableTransmission	:= TRUE;
//ModbusStartTrigger(clk := b_EnableTransmission);

Databuffer[0]	:= OperatingPoint.OperatingMode;	//set operating mode for write
Databuffer[1]	:= 3;								//enable write registers

MBMaster.WriteRegs ( 
					UnitID 		:= 	HeatPumpID,
					Quantity 	:= 	2,
					MBAddr		:=	7200,
					cbLength 	:= 	4,
					pMemoryAddr	:=	ADR(Databuffer),
					Execute		:=	ModbusStartTrigger.Q,
					Timeout		:=	T#250MS,		
					Busy		=>	b_MBBusy,
					Error 		=>	b_MBerr,
					);
				

TransmissionDoneTrigger(clk := b_MBBusy);

IF TransmissionDoneTrigger.q THEN
	IF NOT b_MBerr THEN
				
		//done, preset for next step
		b_EnableTransmission := FALSE;
		ModbusStartTrigger(clk := b_EnableTransmission);
		MBRetryCount := 0;
		sfctip := TRUE;
	ELSE
		MBRetryCount := MBRetryCount + 1;
		b_EnableTransmission	:= FALSE;
		
		//if comm fails 5 times in a row. system is unusable
		IF MBRetryCount > 5 THEN
			get.HeatPumpState := eHeatpumpState.ERROR;
			get.Events.b_CommError := TRUE;
		END_IF
	END_IF
END_IF
END_ACTION

ACTION aWriteSetpoint:

CASE OperatingPoint.OperatingMode OF				//Update setpoint depending on mode
	eHeatPumpMode.Cooling:
		Databuffer[0]	:= REAL_TO_WORD(LIMIT(50, ((Operatingpoint.Setpoint)*10), 230));
		Databuffer[1]	:= REAL_TO_WORD(Get.HeatpumpData.r_SetpointHeating*10);
	eHeatPumpMode.Heating:
		Databuffer[0]	:= REAL_TO_WORD(Get.HeatpumpData.r_SetpointCooling*10);
		Databuffer[1]	:= REAL_TO_WORD(LIMIT(250, ((Operatingpoint.Setpoint)*10), 550));
	eHeatPumpMode.Standby:
		Databuffer[0]	:= REAL_TO_WORD(Get.HeatpumpData.r_SetpointCooling*10);
		Databuffer[1]	:= REAL_TO_WORD(Get.HeatpumpData.r_SetpointHeating*10);	
END_CASE

MBMaster.WriteRegs (
		UnitID 		:= 	HeatPumpID,
		Quantity 	:= 	2,
		MBAddr		:=	7203,
		cbLength 	:= 	4,
		pMemoryAddr	:=	ADR(Databuffer),
		Execute		:=	ModbusStartTrigger.Q,
		Timeout		:=	T#250MS,		
		Busy		=>	b_MBBusy,
		Error 		=>	b_MBerr,
);


TransmissionDoneTrigger(clk := b_MBBusy);

IF TransmissionDoneTrigger.q THEN
	IF NOT b_MBerr THEN
		//done, preset for next step

		MBRetryCount := 0;
		sfctip := TRUE;
	ELSE
		MBRetryCount := MBRetryCount + 1;
		b_EnableTransmission	:= FALSE;
		
		//if comm fails 5 times in a row. system is unusable
		IF MBRetryCount > 5 THEN
			get.HeatPumpState := eHeatpumpState.ERROR;
			get.Events.b_CommError := TRUE;
		END_IF
	END_IF
END_IF
END_ACTION

ACTION ContinousActions:
//sfctip := False;
ModbusRetryTimer(in:= NOT (ModbusRetryTimer.Q OR ResetRetryTimer));
ModbusStartTrigger(clk := ModbusRetryTimer.q);

//for initial use, get notice if 1 packet fails
IF MBRetryCount > 1 THEN
	get.Events.b_CommWarning := TRUE;
END_IF

//ResetRetryTimer := FALSE;
END_ACTION

METHOD ParseHeatPumpErrors : BOOL
VAR_INPUT
	w_Alarms1	:	WORD;
	w_Alarms2	:	WORD;
	w_Alarms3	:	WORD;
	w_Alarms4	:	WORD;
	w_Alarms5	:	WORD;
	w_Alarms6	:	WORD;
	w_Alarms7	:	WORD;
END_VAR		
VAR
	
END_VAR

VAR_IN_OUT
	get	:	ST_HeatpumpGet;	
END_VAR
get.events.b_ProbeError		:=	WORD_TO_BOOL(w_Alarms3) OR WORD_TO_BOOL(w_Alarms4) OR w_Alarms5.0;

get.events.b_PressureError		:=	w_Alarms1.0 OR	//E001: High Pressure
									w_Alarms1.1 OR //E002: Low Pressure
									w_Alarms2.3;	//E020: Inverted Pressure Transducers


get.events.b_CompressorError	:=	w_Alarms1.2 OR //E003: Compressor overheated
									w_Alarms1.7 OR //E008: Compressor underspeed
									w_Alarms1.8 OR	//E009: High disch temp
									w_Alarms1.12 OR //E013: Comp2 Overheated
									w_Alarms2.2 OR	//E019: CP2 High disch temp
									w_Alarms2.6 OR	//E023: Comp3 Overheated
									w_Alarms5.1 OR //'E801: Link Inverter1',
									w_Alarms5.2 OR //'E802: Link Inverter2',
									w_Alarms5.3 OR //'E803: Link Inverter3',
									w_Alarms5.4 OR //'E851: HWfault Inverter1',
									w_Alarms5.5 OR //'E852: HWfault Inverter2',
									w_Alarms5.6 OR //'E853: HWfault Inverter3',
									w_Alarms5.7 OR //'E861: OverCurrent Inv1',
									w_Alarms5.8 OR //'E862: OverCurrent Inv2',
									w_Alarms5.9 OR //'E863: OverCurrent Inv3',
									w_Alarms5.10 OR //'E871: High Temp Inv1',
									w_Alarms5.11 OR //'E872: High Temp Inv2',
									w_Alarms5.12 OR //'E873: High Temp Inv3',
									w_Alarms5.13 OR //'E881: Bad Voltage Inv1',
									w_Alarms5.14 OR //'E882: Bad Voltage Inv2',
									w_Alarms5.15 OR //'E883: Bad Voltage Inv3',
									w_Alarms6.0 OR //E891: Phase Seq Inv1',
									w_Alarms6.1 OR //'E892: Phase Seq Inv2',
									w_Alarms6.2 OR //'E893: Phase Seq Inv3',
									w_Alarms6.3 OR //'E901: Model err Inv1',
									w_Alarms6.4 OR //'E902: Model err Inv2',
									w_Alarms6.5 OR //'E903: Model err Inv3',
									w_Alarms6.6 OR //'E911: Ovl error Inv1',
									w_Alarms6.7 OR //'E9112: Ovl error Inv2',
									w_Alarms6.8 OR //'E913: Ovl error Inv3',
									w_Alarms6.9 OR //'E921: Overc PFC Inv1',
									w_Alarms6.10 OR //'E922: Overc PFC Inv2',
									w_Alarms6.11 OR //'E923: Overc PFC Inv3',
									w_Alarms6.12 OR //'E931: Int Com ERR Inv1',
									w_Alarms6.13 OR //'E932: Int Com ERR Inv2',
									w_Alarms6.14 OR //'E933: Int Com ERR Inv3',
									w_Alarms6.15 OR //'E941: Fault PFC Inv1',
									w_Alarms7.0 OR //E942: Fault PFC Inv2
									w_Alarms7.1 OR //'E943: Fault PFC Inv3',
									w_Alarms7.2 OR //'E951: Probe error Inv1',
									w_Alarms7.3 OR //'E952: Probe error Inv2',
									w_Alarms7.4 OR //'E953: Probe error Inv3',
									w_Alarms7.5 OR //'E961: Abnormal Cond Inv1',
									w_Alarms7.6 OR //'E962: Abnormal Cond Inv2',
									w_Alarms7.7 OR //'E963: Abnormal Cond Inv3',
									w_Alarms7.8 OR //'E971: Inv1 Eeprom Error',
									w_Alarms7.9 OR //'E972: Inv2 Eeprom Error',
									w_Alarms7.10 OR //'E973: Inv3 Eeprom Error',
									w_Alarms7.11;	//E029: CP3 High disch temp

get.events.b_ValveError		:=		w_Alarms2.11; //E041: Incongruent temps;


get.events.b_FanError			:=	w_Alarms1.2 OR //E004: Fan Overheated	
									w_Alarms1.13 OR //E014: Fan2 Overheated 
									w_Alarms2.7;	//E024: Fan3 Overheated					

get.events.b_PumpError			:=	w_Alarms1.5 OR	 	//E006: Lack of flow
									w_Alarms1.15 OR 	//E016: Pump Overheated
									w_Alarms2.9;		//E026: Pump2 Overheated

get.events.b_WaterTempError		:=	w_Alarms2.1 OR	//E018: OverTemperature
									w_Alarms1.4;	//E005: Frost

get.events.b_IOError			:=	w_Alarms2.14 OR 	//E101: IOMod1 Disconnected
									w_Alarms2.15; 		//E102: IOMod2 Disconnected
END_METHOD

ACTION SFCTipReset:
SFCTip := FALSE;
ResetRetryTimer := FALSE;
END_ACTION

END_FUNCTION_BLOCK

// ---- POUs/Objects/CoolingSystem/CoolingStack/FB_HeatPumpSystem.TcPOU
FUNCTION_BLOCK FB_HeatPumpSystem
VAR_INPUT
END_VAR
VAR
	PrimaryHeatpump: FB_Heatpump;
	HeatPumpInitTimeout: TON := (PT := TIME#3S0MS);
END_VAR

VAR_IN_OUT
	b_EnablePower 	: BOOL;
	//r_Setpoint 		: REAL;

//	Faults: ST_CoolingSystemEvents; 
//	HPSSet: ST_CoolingStackSet;
END_VAR

VAR_OUTPUT
	Get : ST_HeatpumpSystemGet;
END_VAR

VAR
	SecondHPPowerOnDelay: 	TON := (PT := TIME#250MS);
	IO	:	FB_HeatpumpSystem_IO;
	MBcommBusy	:	BOOL;
	CommFreeForID	:	BYTE	:= 0;
	CommFreeTimeout	:	TON 	:= (PT := TIME#5s0ms);
	SecondaryHeatPump: FB_Heatpump;
END_VAR

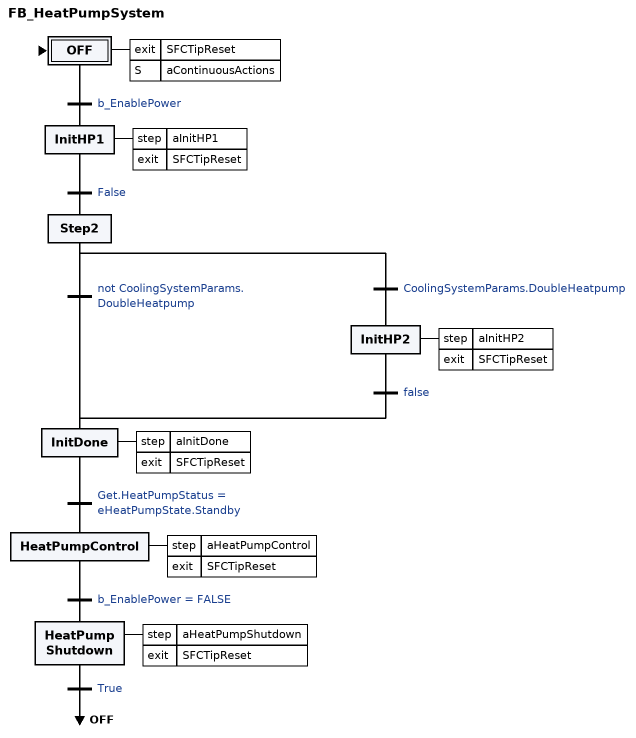
INITIAL_STEP OFF:
    SFCTipReset(P0);  // exit action
    aContinuousActions(S);
END_STEP
TRANSITION FROM OFF TO InitHP1
    := b_EnablePower;
END_TRANSITION
// macro InitHeatpumps begins
STEP InitHP1:
    aInitHP1(N);  // step action
    SFCTipReset(P0);  // exit action
END_STEP
TRANSITION FROM InitHP1 TO Step2
    := False;
END_TRANSITION
STEP Step2:
END_STEP
TRANSITION FROM Step2 TO InitDone
    := not CoolingSystemParams.DoubleHeatpump;
END_TRANSITION
TRANSITION FROM Step2 TO InitHP2
    := CoolingSystemParams.DoubleHeatpump;
END_TRANSITION
STEP InitHP2:
    aInitHP2(N);  // step action
    SFCTipReset(P0);  // exit action
END_STEP
TRANSITION FROM InitHP2 TO InitDone
    := false;
END_TRANSITION
STEP InitDone:
    aInitDone(N);  // step action
    SFCTipReset(P0);  // exit action
END_STEP
TRANSITION FROM InitDone TO HeatPumpControl
    := Get.HeatPumpStatus = eHeatPumpState.Standby;
END_TRANSITION
STEP HeatPumpControl:
    aHeatPumpControl(N);  // step action
    SFCTipReset(P0);  // exit action
END_STEP
TRANSITION FROM HeatPumpControl TO HeatPumpShutdown
    := b_EnablePower = FALSE;
END_TRANSITION
STEP HeatPumpShutdown:
    aHeatPumpShutdown(N);  // step action
    SFCTipReset(P0);  // exit action
END_STEP
TRANSITION FROM HeatPumpShutdown TO OFF
    := True;
END_TRANSITION

ACTION aContinuousActions:
IO(b_EnablePower := b_enablePower);

Get.PrimaryHeatpumpGet REF=PrimaryHeatPump.get;
Get.SecondaryHeatpumpGet REF=SecondaryHeatPump.get;

get.HeatPumpStatus := get.PrimaryHeatpumpGet.HeatPumpState;
END_ACTION

ACTION aHeatPumpControl:

//500ms trigger to switch MB bus ownership to next heatpump
CommFreeTimeout(in := NOT CommFreeTimeout.Q);
IF CommFreeTimeout.Q OR (not MBCommBusy) THEN
	CommFreeForID := (CommFreeForID+1) MOD 2;
END_IF

//FB returns MBCommBusy to indicate when status update is done. Could be used for optimized RW speed
//Not used at this moment

PrimaryHeatPump(ACPowerStatus := b_EnablePower, MBFree := (CommFreeForID=0), MBcommBusy => MBcommBusy);
//IF CoolingSystemParams.DoubleHeatpump THEN
//	HeatPumps[2](ACPowerStatus := b_EnablePower, MBFree := (CommFreeForID=1));
//END_IF
END_ACTION

ACTION aHeatPumpShutdown:
Get.HeatPumpStatus := eHeatPumpState.OFF;
END_ACTION

ACTION aInitDone:

get.HeatPumpStatus := eHeatPumpState.Standby;
END_ACTION

ACTION aInitHP1:

IF Coolingsystemparams.DoubleHeatpump THEN
	SecondaryHeatpump(ACPowerStatus := FALSE, MBFree := FALSE);
END_IF

IF PrimaryHeatpump.get.HeatPumpState <= eHeatpumpstate.Initializing THEN
	PrimaryHeatpump(ACPowerStatus := b_EnablePower, MBFree := TRUE);
ELSIF PrimaryHeatpump.get.HeatPumpState = eHeatpumpstate.Standby THEN
	PrimaryHeatpump(ACPowerStatus := b_EnablePower, MBFree := FALSE);
	SFCTip := TRUE;
END_IF
END_ACTION

ACTION aInitHP2:


IF SecondaryHeatpump.get.HeatPumpState = eHeatpumpstate.Initializing THEN
	SecondaryHeatpump(ACPowerStatus := b_EnablePower, MBFree := TRUE);
ELSIF SecondaryHeatpump.get.HeatPumpState = eHeatpumpstate.Standby THEN
	SecondaryHeatpump(ACPowerStatus := b_EnablePower, MBFree := FALSE);
	SFCTip := TRUE;
END_IF
END_ACTION

ACTION aPowerControl:
IO(b_EnablePower := b_enablePower);
END_ACTION

METHOD EMStop : BOOL
VAR_INPUT
END_VAR
EMstop := PrimaryHeatpump.emstop() and SecondaryHeatpump.emstop();
END_METHOD

METHOD GetDiagnostics 
VAR_IN_OUT
	AddError		: ARRAY [*] OF FB_AddErrorST;
	a_ActiveEvents	: ARRAY [*] OF ST_ErrorStruct;
	w_Index			: WORD;
END_VAR

VAR_OUTPUT
	b_errorActive	: BOOL;
	b_warningActive	: BOOL;
END_VAR

VAR
	by_errCt	: BYTE;
	by_warnCt	: BYTE;
	w_ID		: WORD;
END_VAR

//check if this call works:
PrimaryHeatpump.GetDiagnostics(AddError := AddError, a_ActiveEvents := a_ActiveEvents, w_Index := w_Index, b_errorActive => b_errorActive, b_warningActive => b_warningActive);

//not in use
//Heatpumps[2].GetDiagnostics(AddError := AddError, a_ActiveEvents := a_ActiveEvents, w_Index := w_Index, b_errorActive => b_errorActive, b_warningActive => b_warningActive);
END_METHOD

METHOD Reset : BOOL
VAR_INPUT
END_VAR
Reset := PrimaryHeatpump.Reset() and SecondaryHeatpump.Reset();
END_METHOD

ACTION SFCTipReset:
SFCTip := FALSE;
END_ACTION

METHOD WriteSetpoint : BOOL
VAR_INPUT
	OperatingMode	:	eHeatpumpMode;
	SetPoint		: 	REAL;
END_VAR
PrimaryHeatpump.WriteSetpoint(OperatingMode := OperatingMode, SetPoint := Setpoint);

//This method will also contain potential master/slave temperature differentials and other differences between heatpumps
//Heatpumps[2].WriteSetpoint(OperatingMode := OperatingMode);
END_METHOD

END_FUNCTION_BLOCK

// ---- POUs/Objects/CoolingSystem/CoolingStack/FB_Heatpumpsystem_IO.TcPOU
FUNCTION_BLOCK FB_Heatpumpsystem_IO
VAR_INPUT
	b_EnablePower	:	BOOL;
END_VAR

VAR_OUTPUT
	PrimaryHeatpump_EnablePower	AT %Q* :	BOOL;
	SecondaryHeatpump_EnablePower	AT %Q* :	BOOL;
END_VAR
VAR
	PowerOnDelay: TON := (PT := TIME#100MS);
END_VAR


//heatpump 2 is enabled with a delay to limit inrush
PrimaryHeatpump_EnablePower := b_EnablePower;
IF CoolingSystemParams.DoubleHeatpump THEN
	PowerOnDelay(IN := b_EnablePower);
	SecondaryHeatpump_EnablePower := PowerOnDelay.Q;
END_IF

END_FUNCTION_BLOCK

// ---- POUs/Objects/CoolingSystem/FB_CoolingSystem.TcPOU
FUNCTION_BLOCK FB_CoolingSystem

VAR
	ConditioningMode			:	eConditioningStates;
	
	ControlData					:	ST_CoolingSystem_Control;
	ConditioningRequirements	:	ST_ConditioningRequirements;
	
	BatteryConditioningSFC		:	FB_BatteryConditioningSFC;
	DehumSFC					:	FB_DehumidifySFC;
	EnclosureConditioningSFC	:	FB_EnclosureConditioningSFC;
	PowerModeConditioningSFC	:	FB_PowerModeConditioningSFC;
	
	Heatpumps					:	FB_HeatPumpSystem;
	
	FB_IO						:	FB_CoolingSystem_IO;
END_VAR;

VAR_OUTPUT
	Get: ST_CoolingSystemGet;		//Various cooling sytem data for logging
END_VAR

VAR_IN_OUT
//Inputs
	//From Powerstack Inverter cooling request
	by_SetCooling			:	BYTE;	//Inverter request cooling. 0=none, 1=startup only, 2=power delivery mode
	b_InverterRunning		: 	BOOL;	//True if inverter is modulating, used as determine when pumps may shutdown
	r_InverterTemperature	:	REAL;	//Inverter Internal temperature
	r_InverterPowerLevel	:	REAL;	//Inverter output power (kVA/kW) to determine expected system heat generation
	r_CMSTemperature		:	REAL;	//Combined CMS temperature
	
	//Internal power supply status
	b_24v_Available			:	BOOL;	//from FB_ips, 24V online
	b_400v_Available 		:	BOOL;	//from FB_ips, 400vac online

	//From BMS
	r_BMSAverageBattTemp	:	REAL;	//from FB_BMS, average battery temperature
	r_BMSMaxBattTemp		:	REAL;	//from FB_BMS, max battery temperature (may not be needed)
	
	//From Enclosure
	r_EnclosureHumidity		:	REAL;	//from FB_enclosure
	r_EnclosureTemperature	:	REAL;	//from FB_enclosure
	
//Outputs
	//To powerstack: 
	by_PSCoolingPowerMode	: 	BYTE; 	//Allowed operating mode for inverter. 0: no modulating allowed, 1: modulating allowed, no power delivery, 2:inverter power delivery allowed.
	IPSDemand : ST_PowerDemand;			//to FB_IPS, power requirements for cooling system
END_VAR

//Exchange external data into datastruct (for simpler passing around within the cooling system)
by_PSCoolingPowerMode 					:= 	ConditioningRequirements.by_PSCoolingPowerMode;
ConditioningRequirements.by_SetCooling 	:= 	by_SetCooling;
ControlData.b_InverterRunning			:=	b_InverterRunning;
ControlData.r_BMSBatteryTemperature 	:= 	r_BMSAverageBattTemp;
ControlData.R_BMSMaxBatteryTemperature	:=	r_BMSMaxBattTemp;
ControlData.r_EnclosureHumidity			:=	r_EnclosureHumidity;
ControlData.r_EnclosureTemperature		:=	r_EnclosureTemperature;
ControlData.r_InverterTemperature		:=	r_InverterTemperature;
ControlData.r_OutputPowerLevel			:=	r_InverterPowerLevel;
ControlData.b_24V_Available				:=	b_24V_Available;
ControlData.b_400v_Available			:=	b_400V_Available;
	
//Call local IO functionblock	
FB_IO(IO := ControlData, Events := get.Events);

//Call standby climate monitors for Battery and enclosure 
BatteryIdleMonitor(Control := ControlData, ConditioningRequirements := ConditioningRequirements);
EnclosureIdleMonitor(Control := ControlData, ConditioningRequirements := ConditioningRequirements);

//Determine which SFC to start, based on current status and priority. 
SetConditioningMode();

//Call climate control SFC's
EnclosureConditioningSFC(IPSDemand := IPSDemand, Control := ControlData, ConditioningRequirements := ConditioningRequirements, Get := Get);
BatteryConditioningSFC	(IPSDemand := IPSDemand, Control := ControlData, ConditioningRequirements := ConditioningRequirements, Get := Get);
PowerModeConditioningSFC(IPSDemand := IPSDemand, Control := ControlData, ConditioningRequirements := ConditioningRequirements, Get := Get);
DehumSFC				(IPSDemand := IPSDemand, Control := ControlData, ConditioningRequirements := ConditioningRequirements, Get := Get);

//These only work as long as there is external 400VAC (as HVDC is shutdown). So no real need to shutdown imo.
(*
IF ConditioningMode = eConditioningStates.EMSTOP THEN
	IF ControlData.r_InverterTemperature < CoolingSystemParams.EMSTOPInverterIdleShutdownTemp AND
		ControlData.R_BMSMaxBatteryTemperature < CoolingSystemParams.EMSTOPBatteryShutdownTemp THEN
			//Shutdown 24V coolingdown loop activated in EMSTOP method to prevent UPS battery drain
			ControlData.b_DCPumpEnable 				:= FALSE;
			ControlData.b_CloseInverterLoopValve	:= FALSE;
			ControlData.b_CloseBatteryLoopValve 	:= FALSE;
			ControlData.b_CloseFancoilLoopValve 	:= FALSE;
	END_IF
END_IF
*)

//Call Heatpump FB
HeatPumps(b_EnablePower := ControlData.b_HeatPumpPowerEnable);
get.HeatPumpSystemGet REF= Heatpumps.Get;
Heatpumps.WriteSetpoint(OperatingMode := ControlData.e_HeatpumpMode, Setpoint := ControlData.r_HeatPumpSetpoint);
get.HeatPumpStatus := get.HeatPumpSystemGet.HeatPumpStatus;

METHOD BatteryIdleMonitor : BOOL
VAR_IN_OUT
	Control 							:	ST_CoolingSystem_Control;
	ConditioningRequirements 	: 	ST_ConditioningRequirements;
END_VAR

//Battery cooling is triggered by the set Max temp. System then cools down to the midway point between Battery max and min.
//Battery heating is triggered by the set Min temp. System then warms up to the midway point between Battery max and min.
//Halfway points are chosen to limit Battery conditioning frequency

CASE ConditioningRequirements.Battery OF
	eConditioningRequirement.None:
		IF Control.r_BMSBatteryTemperature > CoolingSystemParams.BatteryIdleTempMax THEN
			ConditioningRequirements.Battery := eConditioningRequirement.Cooling;
		ELSIF Control.r_BMSBatteryTemperature < CoolingSystemParams.BatteryIdleTempMin THEN
			ConditioningRequirements.Battery := eConditioningRequirement.Heating;
		END_IF
		
	eConditioningRequirement.Heating:
		IF Control.r_BMSBatteryTemperature >= (CoolingSystemParams.BatteryIdleTempMin+CoolingSystemParams.BatteryIdleTempMax)/2 THEN
			ConditioningRequirements.Battery := eConditioningRequirement.None;
		END_IF
		
	eConditioningRequirement.Cooling:
		IF Control.r_BMSBatteryTemperature <= (CoolingSystemParams.BatteryIdleTempMin+CoolingSystemParams.BatteryIdleTempMax)/2 THEN
			ConditioningRequirements.Battery := eConditioningRequirement.None;
		END_IF
END_CASE
END_METHOD

METHOD EMSTOP : BOOL
VAR_INPUT
END_VAR

ConditioningMode := eConditioningStates.EMSTOP;

EnclosureConditioningSFC.SFCEnable(Enable:= FALSE);
BatteryConditioningSFC.SFCEnable(Enable:= FALSE);
PowerModeConditioningSFC.SFCEnable(Enable:= FALSE);
DehumSFC.SFCEnable(Enable:= FALSE);

//Keep 24V cooling enabled
ControlData.b_DCPumpEnable 				:= TRUE;
ControlData.b_CloseInverterLoopValve	:= FALSE;
ControlData.b_CloseBatteryLoopValve 	:= FALSE;
ControlData.b_CloseFancoilLoopValve 	:= TRUE;

ControlData.b_ACPumpEnable 				:= FALSE;
ControlData.b_HeatPumpPowerEnable 		:= FALSE;


ControlData.b_DCFancoilEnable 			:= FALSE;

EMSTOP := Heatpumps.EMStop();
END_METHOD

METHOD EnclosureIdleMonitor : BOOL
VAR_IN_OUT
	Control 							:	ST_CoolingSystem_Control;
	ConditioningRequirements 	: 	ST_ConditioningRequirements;
END_VAR

VAR
	alpha					: REAL;
END_VAR

//Calculate system dewpoint
alpha := LN(Control.r_EnclosureHumidity/100)+(17.625*Control.r_EnclosureTemperature/(243.12+Control.r_EnclosureTemperature));
Control.r_CurrentEnclosureDewPoint := 243.12*alpha/(17.625-alpha);


//Enclosure cooling is triggered by the set Max temp. System then cools down to the midway point between Enclosure max and Battery max.
//Enclosure heating is triggered by the highest temp between Enclosure min and current dew point. The highest is used to compensate for high dewpoints.
//Enclosure heating is done if the halfwaypoint between battery temp min and enclosure temp min.
//Halfway points are chosen to prevent prolonged conditioning runs
CASE ConditioningRequirements.Enclosure OF
	eConditioningRequirement.None:
		IF Control.r_EnclosureTemperature > CoolingSystemParams.EnclosureIdleTempMax THEN
			ConditioningRequirements.Enclosure := eConditioningRequirement.Cooling;
		ELSIF Control.r_EnclosureTemperature < MAX(CoolingSystemParams.EnclosureIdleTempMin, Control.r_CurrentEnclosureDewPoint) THEN
			ConditioningRequirements.Enclosure := eConditioningRequirement.Heating;
		END_IF
		
	eConditioningRequirement.Heating:
		IF Control.r_EnclosureTemperature < (CoolingSystemParams.EnclosureIdleTempMin+CoolingSystemParams.BatteryIdleTempMin)/2 THEN
			ConditioningRequirements.Enclosure := eConditioningRequirement.None;
		END_IF
		
	eConditioningRequirement.Cooling:
		IF Control.r_EnclosureTemperature < (CoolingSystemParams.EnclosureIdleTempMax+CoolingSystemParams.BatteryIdleTempMax)/2 THEN
			ConditioningRequirements.Enclosure := eConditioningRequirement.None;
		END_IF
END_CASE
END_METHOD

METHOD GetDiagnostics 
VAR_IN_OUT
	AddError		: ARRAY [*] OF FB_AddErrorST;
	a_ActiveEvents	: ARRAY [*] OF ST_ErrorStruct;
	w_Index			: WORD;
END_VAR

VAR_OUTPUT
	b_errorActive	: BOOL;
	b_warningActive	: BOOL;
END_VAR

VAR
	by_errCt	: BYTE;
	by_warnCt	: BYTE;
	w_ID		: WORD;
END_VAR
	(*Battery loop valve stuck*)	AddError[w_Index](
			in_b_ErrorTrig			:= Get.Events.b_BattLoopValveStuck,
			out_ST_Error			:= a_ActiveEvents[w_Index],
			w_ID					:= 1 + w_ID,
			s_Message				:= 'Battery cooling loop valve fault',
			e_sev					:= eSeverity.NormalShutdown,	
			in_b_AutoClear			:= FALSE,
			//in_e_ErrAckAccess		:= TRUE,
			);
		IF AddError[w_Index].b_out THEN by_errCt := by_errCt + 1; END_IF;
		w_Index := w_Index +1;
		
	(*Fancoil loop valve stuck*)	AddError[w_Index](
			in_b_ErrorTrig			:= Get.Events.b_BattLoopValveStuck,
			out_ST_Error			:= a_ActiveEvents[w_Index],
			w_ID					:= 2 + w_ID,
			s_Message				:= 'Fancoil cooling loop valve fault',
			e_sev					:= eSeverity.NormalShutdown,	
			in_b_AutoClear			:= FALSE,
			//in_e_ErrAckAccess		:= TRUE,
			);
		IF AddError[w_Index].b_out THEN by_errCt := by_errCt + 1; END_IF;
		w_Index := w_Index +1;
	
	(*Inverter loop valve stuck*)	AddError[w_Index](
			in_b_ErrorTrig			:= Get.Events.b_InverterLoopValveStuck,
			out_ST_Error			:= a_ActiveEvents[w_Index],
			w_ID					:= 3 + w_ID,
			s_Message				:= 'Inverter cooling loop valve fault',
			e_sev					:= eSeverity.QuickShutdown,	
			in_b_AutoClear			:= FALSE,
			//in_e_ErrAckAccess		:= TRUE,
			);
		IF AddError[w_Index].b_out THEN by_errCt := by_errCt + 1; END_IF;
		w_Index := w_Index +1;
		
	(*Inverter cooling error*)	AddError[w_Index](
			in_b_ErrorTrig			:= Get.Events.b_InverterCoolingLoopError,
			out_ST_Error			:= a_ActiveEvents[w_Index],
			w_ID					:= 4 + w_ID,
			s_Message				:= 'Inverter cooling loop failed',
			e_sev					:= eSeverity.QuickShutdown,	
			in_b_AutoClear			:= FALSE,
			//in_e_ErrAckAccess		:= TRUE,
			);
		IF AddError[w_Index].b_out THEN by_errCt := by_errCt + 1; END_IF;
		w_Index := w_Index +1;
		
	(*Heatpump Warning*)		AddError[w_Index](
			in_b_ErrorTrig			:= Get.Events.b_HeatpumpWarning,
			out_ST_Error			:= a_ActiveEvents[w_Index],
			w_ID					:= 5 + w_ID,
			s_Message				:= 'Heatpump warning',
			e_sev					:= eSeverity.Warning,	
			in_b_AutoClear			:= FALSE,
			//in_e_ErrAckAccess		:= TRUE,
			);
		IF AddError[w_Index].b_out THEN by_warnCt := by_warnCt + 1; END_IF;
		w_Index := w_Index +1;		
	
	(*Heatpump inoperative*)		AddError[w_Index](
			in_b_ErrorTrig			:= Get.Events.b_HeatPumpError ,
			out_ST_Error			:= a_ActiveEvents[w_Index],
			w_ID					:= 6 + w_ID,
			s_Message				:= 'Heatpump inoperative',
			e_sev					:= eSeverity.NormalShutdown,	
			in_b_AutoClear			:= FALSE,
			//in_e_ErrAckAccess		:= TRUE,
			);
		IF AddError[w_Index].b_out THEN by_errCt := by_errCt + 1; END_IF;
		w_Index := w_Index +1;
		
	(*400V fuse failure*)			AddError[w_Index](
			in_b_ErrorTrig			:= Get.Events.b_CoolingSystemFuseFailure,
			out_ST_Error			:= a_ActiveEvents[w_Index],
			w_ID					:= 7 + w_ID,
			s_Message				:= 'Cooling system 400V fuse fault',
			e_sev					:= eSeverity.QuickShutdown,	
			in_b_AutoClear			:= FALSE,
			//in_e_ErrAckAccess		:= TRUE,
			);
		IF AddError[w_Index].b_out THEN by_errCt := by_errCt + 1; END_IF;
		w_Index := w_Index +1;
		
	(*Coolant pressure lost*)		AddError[w_Index](
			in_b_ErrorTrig			:= Get.Events.b_CoolingLoopIdlePressureError,
			out_ST_Error			:= a_ActiveEvents[w_Index],
			w_ID					:= 8 + w_ID,
			s_Message				:= 'Cooling system pressure fault',
			e_sev					:= eSeverity.NormalShutdown,	
			in_b_AutoClear			:= FALSE,
			//in_e_ErrAckAccess		:= TRUE,
			);
		IF AddError[w_Index].b_out THEN by_errCt := by_errCt + 1; END_IF;
		w_Index := w_Index +1;	
	
	(*Coolant pressure low*)		AddError[w_Index](
			in_b_ErrorTrig			:= Get.Events.b_CoolingLoopIdlePressureWarning,
			out_ST_Error			:= a_ActiveEvents[w_Index],
			w_ID					:= 9 + w_ID,
			s_Message				:= 'Cooling system pressure warning',
			e_sev					:= eSeverity.Warning,	
			in_b_AutoClear			:= FALSE,
			//in_e_ErrAckAccess		:= TRUE,
			);
		IF AddError[w_Index].b_out THEN by_WarnCt := by_WarnCt + 1; END_IF;
		w_Index := w_Index +1;	

		
		
//check if this call works:
Heatpumps.GetDiagnostics(AddError := AddError, a_ActiveEvents := a_ActiveEvents, w_Index := w_Index, b_errorActive => b_errorActive, b_warningActive => b_warningActive);
END_METHOD

METHOD ProcessOutputData : BOOL
VAR_INPUT
END_VAR
END_METHOD

METHOD Reset : BOOL
VAR
	b_ActiveErrors		:	BOOL;
	b_ActiveWarnings	:	BOOL;
END_VAR
Reset := FALSE;

//Set in SFC, but will not self clear. Reset at this point. It will fail again when restarting
//No way of testing it prior to that point
get.Events.b_InverterCoolingLoopError := FALSE;


b_ActiveErrors := 	Get.Events.b_BattLoopValveStuck OR
					Get.Events.b_CoolingLoopIdlePressureError OR
					Get.Events.b_InverterCoolingLoopError OR
					Get.Events.b_CoolingSystemFuseFailure OR
					Get.Events.b_FancoilLoopValveStuck OR
					Get.Events.b_HeatPumpError OR
					Get.Events.b_InverterLoopValveStuck;

IF NOT b_ActiveErrors THEN
	IF ConditioningMode = eConditioningStates.EMSTOP THEN
		ConditioningMode := eConditioningStates.OFF;
	END_IF
	
	Reset := Heatpumps.Reset();
END_IF;
END_METHOD

METHOD SetConditioningMode : BOOL
VAR_INPUT
END_VAR
IF ConditioningMode <> eConditioningStates.EMSTOP THEN
	//Determine which SFC should be active, halt all others.
	IF (ConditioningRequirements.by_SetCooling = 2) OR (PowerModeConditioningSFC.SFCActive) THEN
		ConditioningMode := eConditioningStates.InverterPowerMode;		
	ELSIF (ConditioningRequirements.Battery <> eConditioningRequirement.None) OR (BatteryConditioningSFC.SFCActive) THEN
		ConditioningMode := eConditioningStates.BatteryConditioning;
	ELSIF ConditioningRequirements.Dehum OR (DehumSFC.SFCActive) THEN
		ConditioningMode := eConditioningStates.DeHum;
	ELSIF ConditioningRequirements.by_setCooling = 1	THEN
		//If this is true, no AC conditioning mode is required but the inverter is still asking for low power cooling. This is ZPTinit mode
		//After executing this code once, the next iterations will run the first if statement until finished 
		ConditioningMode := eConditioningStates.InverterZPTStartup;
	ELSIF ConditioningRequirements.Enclosure <> eConditioningRequirement.None  OR (EnclosureConditioningSFC.SFCActive) THEN
		ConditioningMode := eConditioningStates.EnclosureConditioning;
	ELSE
		ConditioningMode := eConditioningStates.OFF;
	END_IF
END_IF

//SFC stuck in Init=true unless that conditioningmode is active
BatteryConditioningSFC.SFCEnable(Enable:= (ConditioningMode = eConditioningStates.BatteryConditioning));
DehumSFC.SFCEnable(Enable:=  (ConditioningMode = eConditioningStates.DeHum));
EnclosureConditioningSFC.SFCEnable(Enable:=  (ConditioningMode = eConditioningStates.EnclosureConditioning));
PowerModeConditioningSFC.SFCEnable(Enable:=  ((ConditioningMode = eConditioningStates.InverterPowerMode ) OR
									   		(ConditioningMode = eConditioningStates.InverterZPTStartup) ));
END_METHOD

END_FUNCTION_BLOCK

// ---- POUs/Objects/CoolingSystem/SFC/FB_BatteryConditioningSFC.TcPOU
FUNCTION_BLOCK FB_BatteryConditioningSFC
VAR_IN_OUT
	IPSDemand					:	ST_PowerDemand;
	ConditioningRequirements	: 	ST_ConditioningRequirements;
	Control						:	ST_CoolingSystem_Control;
	Get							:	ST_CoolingSystemGet;	
END_VAR



VAR_OUTPUT
	SFCCurrentStep	:	STRING;
END_VAR
VAR_OUTPUT
	SFCActive	:	BOOL;
END_VAR

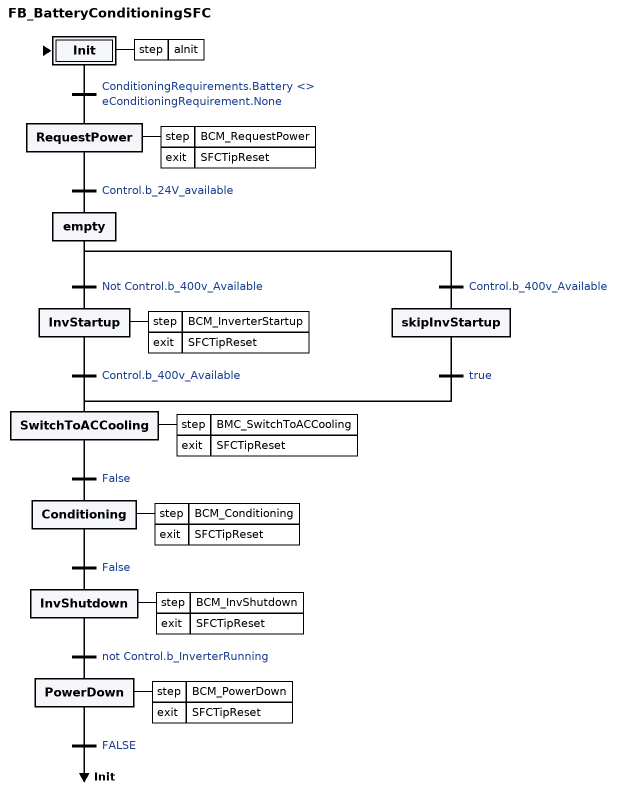
INITIAL_STEP Init:
    aInit(N);  // step action
END_STEP
TRANSITION FROM Init TO RequestPower
    := ConditioningRequirements.Battery <> eConditioningRequirement.None;
END_TRANSITION
STEP RequestPower:
    BCM_RequestPower(N);  // step action
    SFCTipReset(P0);  // exit action
END_STEP
TRANSITION FROM RequestPower TO empty
    := Control.b_24V_available;
END_TRANSITION
STEP empty:
END_STEP
TRANSITION FROM empty TO InvStartup
    := Not Control.b_400v_Available;
END_TRANSITION
STEP InvStartup:
    BCM_InverterStartup(N);  // step action
    SFCTipReset(P0);  // exit action
END_STEP
TRANSITION FROM InvStartup TO SwitchToACCooling
    := Control.b_400v_Available;
END_TRANSITION
TRANSITION FROM empty TO skipInvStartup
    := Control.b_400v_Available;
END_TRANSITION
STEP skipInvStartup:
END_STEP
TRANSITION FROM skipInvStartup TO SwitchToACCooling
    := true;
END_TRANSITION
STEP SwitchToACCooling:
    BMC_SwitchToACCooling(N);  // step action
    SFCTipReset(P0);  // exit action
END_STEP
TRANSITION FROM SwitchToACCooling TO Conditioning
    := False;
END_TRANSITION
STEP Conditioning:
    BCM_Conditioning(N);  // step action
    SFCTipReset(P0);  // exit action
END_STEP
TRANSITION FROM Conditioning TO InvShutdown
    := False;
END_TRANSITION
STEP InvShutdown:
    BCM_InvShutdown(N);  // step action
    SFCTipReset(P0);  // exit action
END_STEP
TRANSITION FROM InvShutdown TO PowerDown
    := not Control.b_InverterRunning;
END_TRANSITION
STEP PowerDown:
    BCM_PowerDown(N);  // step action
    SFCTipReset(P0);  // exit action
END_STEP
TRANSITION FROM PowerDown TO Init
    := FALSE;
END_TRANSITION

ACTION aInit:
SFCActive := False;
END_ACTION

ACTION BCM_Conditioning:

//No real demand for complicated regulation?
//system is off. Just return the average battery temperature to nominal.

//for now just test with fixed setpoints

CASE ConditioningRequirements.Battery OF
	eConditioningRequirement.Cooling:
		Control.e_HeatpumpMode := eHeatpumpmode.Cooling;
		Control.r_HeatPumpSetpoint := 15.0;//minimum adviced battery temperature. Setpoint could be lower, but watch out for inverter condensation.
	eConditioningRequirement.Heating:
		Control.e_HeatpumpMode := eHeatpumpmode.Heating;
		Control.r_HeatPumpSetpoint := 35.0; //minimum heating setpoint
	eConditioningRequirement.None:
		Control.e_HeatpumpMode := eHeatpumpmode.Standby;
		SFCTip := TRUE;
END_CASE

//if coolantpressure drops below startup minimum while inverter is running, shutdown system immediately!
IF 	Control.b_InverterRunning AND
 	(Control.r_CoolantPressure < (CoolingSystemParams.StartupPumpMinimumPressure + Control.r_CoolantIdlePressure)) THEN
		get.Events.b_InverterCoolingLoopError := TRUE;
		ConditioningRequirements.by_PSCoolingPowerMode := 0;
END_IF
END_ACTION

ACTION BCM_Cooldown:

IF ConditioningRequirements.Battery = eConditioningRequirement.Cooling THEN
	Control.b_CloseBatteryLoopValve := FALSE;
	Control.r_HeatPumpSetpoint := 15.0;
ELSIF ConditioningRequirements.Battery = eConditioningRequirement.Heating THEN
	Control.b_CloseBatteryLoopValve := FALSE;
	Control.r_HeatPumpSetpoint := 25.0;
ELSE
	//battery conditioning done, close valve to speed up other conditioning loops
	Control.b_CloseBatteryLoopValve := TRUE;
	IF ConditioningRequirements.Enclosure = eConditioningRequirement.Heating THEN
		Control.r_HeatPumpSetpoint := 25.0;
	ELSIF ConditioningRequirements.Enclosure = eConditioningRequirement.Cooling THEN
		Control.r_HeatPumpSetpoint := 15.0;
	//ELSE
		//if enclosure and battery are ok. Inverter is presumably already cooled down enough. 
		//If not, keep running in current mode for longer
	//	IF PSGet.r_TemperatureMax < CoolingSystemParams.InverterIdleShutdownTemp THEN
		//	ConditioningModeRequired := eConditioningStates.OFF;
		//END_IF
	END_IF	
END_IF
END_ACTION

ACTION BCM_InverterStartup:
Control.b_CloseBatteryLoopValve 	:= TRUE;
Control.b_CloseFancoilLoopValve		:= TRUE;
Control.b_CloseInverterLoopValve	:= FALSE;

Control.b_DCFancoilEnable	:=	FALSE;
//Control.b_ACFancoilEnable	:=	FALSE;

Control.b_DCPumpEnable		:= TRUE;
Control.b_ACPumpEnable		:= FALSE;

Control.b_HeatPumpPowerEnable := FALSE;

//if both are ok, the inverter should have enough flow to start
IF Control.r_CoolantPressure > (CoolingSystemParams.StartupPumpMinimumPressure + Control.r_CoolantIdlePressure) AND Control.b_InverterLoopEnabled THEN
	//Inverter may commence modulating, but no power delivery yet.
	ConditioningRequirements.by_PSCoolingPowerMode := 1;
END_IF
END_ACTION

ACTION BCM_InvShutdown:
Control.b_CloseBatteryLoopValve 	:= TRUE;
Control.b_CloseFancoilLoopValve	:= TRUE;
Control.b_CloseInverterLoopValve	:= FALSE;

Control.b_DCFancoilEnable	:=	FALSE;
//Control.b_ACFancoilEnable	:=	FALSE;

Control.b_DCPumpEnable		:= TRUE;
Control.b_ACPumpEnable		:= FALSE;

Control.b_HeatPumpPowerEnable := FALSE;

//Inverter may shutdown now
ConditioningRequirements.by_PSCoolingPowerMode := 0;
END_ACTION

ACTION BCM_PowerDown:
Control.b_CloseBatteryLoopValve 	:= 	FALSE;
Control.b_CloseFancoilLoopValve	:= 	FALSE;
Control.b_CloseInverterLoopValve	:= 	FALSE;

Control.b_DCFancoilEnable		:=	FALSE;
//Control.b_ACFancoilEnable		:=	FALSE;

Control.b_DCPumpEnable			:= 	FALSE;
Control.b_ACPumpEnable			:= 	FALSE;

Control.b_HeatPumpPowerEnable 	:= 	FALSE;

IPSDemand.b_Demand_24V 			:= FALSE;

Control.e_HeatpumpMode := eHeatpumpMode.Standby; 
SFCActive:= False;
END_ACTION

ACTION BCM_RequestPower:
SFCActive:= True;
IPSDemand.b_Demand_24V := TRUE;
IPSDemand.b_Demand_400V := TRUE;
END_ACTION

ACTION BMC_SwitchToACCooling:
Control.b_DCFancoilEnable 		:= FALSE;
//Control.b_ACFancoilEnable		:= FALSE;


//First enable both pumps to see if AC pump works (by checking pressure increase)
Control.b_ACPumpEnable 			:= TRUE;
Control.b_DCPumpEnable 			:= TRUE;

IF Control.r_CoolantPressure > (CoolingSystemParams.MainPumpMinimumPressure + Control.r_CoolantIdlePressure) THEN
	Control.b_CloseBatteryLoopValve 	:= FALSE;
	Control.b_CloseFancoilLoopValve 	:= FALSE;
	Control.b_CloseBatteryLoopValve 	:= FALSE;
	Control.b_HeatPumpPowerEnable 	:= TRUE;
	Control.b_DCPumpEnable 			:= FALSE;
	Control.e_HeatpumpMode := eHeatpumpmode.Standby;
	Control.r_HeatPumpSetpoint := 18.0;
	SFCTip := TRUE;
END_IF
END_ACTION

METHOD SFCEnable : BOOL
VAR_INPUT
	Enable	:	Bool;
END_VAR
IF Enable THEN
	SFCInit := FALSE;
ELSE
	SFCActive:= FALSE;
	SFCInit := TRUE;
END_IF
END_METHOD

ACTION SFCTipReset:
SFCTip := FALSE;
END_ACTION

END_FUNCTION_BLOCK

// ---- POUs/Objects/CoolingSystem/SFC/FB_DehumidifySFC.TcPOU
FUNCTION_BLOCK FB_DehumidifySFC

VAR_OUTPUT
	SFCCurrentStep	:	STRING;
END_VAR
VAR_IN_OUT
	//IPSState					:	ST_InternalPowerStatus;
	IPSDemand					:	ST_PowerDemand;
	ConditioningRequirements	: 	ST_ConditioningRequirements;
	Control						:	ST_CoolingSystem_Control;
	Get							:	ST_CoolingSystemGet;	
END_VAR
VAR_OUTPUT
	SFCActive	:	BOOL;
END_VAR

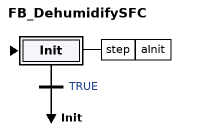
INITIAL_STEP Init:
    aInit(N);  // step action
END_STEP
TRANSITION FROM Init TO Init
    := TRUE;
END_TRANSITION

ACTION aInit:
SFCActive := False;
END_ACTION

METHOD SFCEnable : BOOL
VAR_INPUT
	Enable	:	Bool;
END_VAR
IF Enable THEN
	SFCInit := FALSE;
ELSE
	SFCActive:= FALSE;
	SFCInit := TRUE;
END_IF
END_METHOD

END_FUNCTION_BLOCK

// ---- POUs/Objects/CoolingSystem/SFC/FB_EnclosureConditioningSFC.TcPOU
FUNCTION_BLOCK FB_EnclosureConditioningSFC
VAR_IN_OUT
	//IPSState					:	ST_InternalPowerStatus;
	IPSDemand					:	ST_PowerDemand;
	ConditioningRequirements	: 	ST_ConditioningRequirements;
	Control							:	ST_CoolingSystem_Control;
	Get							:	ST_CoolingSystemGet;	
END_VAR

VAR_OUTPUT
	SFCCurrentStep	:	STRING;
END_VAR
VAR_OUTPUT
	SFCActive	:	BOOL;
END_VAR

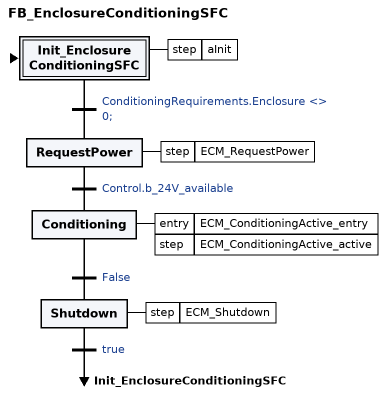
INITIAL_STEP Init_EnclosureConditioningSFC:
    aInit(N);  // step action
END_STEP
TRANSITION FROM Init_EnclosureConditioningSFC TO RequestPower
    := ConditioningRequirements.Enclosure <> 0;
END_TRANSITION
STEP RequestPower:
    ECM_RequestPower(N);  // step action
END_STEP
TRANSITION FROM RequestPower TO Conditioning
    := Control.b_24V_available;
END_TRANSITION
STEP Conditioning:
    ECM_ConditioningActive_entry(P1);  // entry action
    ECM_ConditioningActive_active(N);  // step action
END_STEP
TRANSITION FROM Conditioning TO Shutdown
    := False;
END_TRANSITION
STEP Shutdown:
    ECM_Shutdown(N);  // step action
END_STEP
TRANSITION FROM Shutdown TO Init_EnclosureConditioningSFC
    := true;
END_TRANSITION

ACTION aInit:
SFCActive := False;
END_ACTION

ACTION ECM_ConditioningActive_active:
IF ConditioningRequirements.Enclosure = 0 THEN
	SFCTip := TRUE;
END_IF
END_ACTION

ACTION ECM_ConditioningActive_entry:
Control.b_CloseBatteryLoopValve 	:= 	FALSE;
Control.b_CloseFancoilLoopValve 	:= 	FALSE;
Control.b_CloseInverterLoopValve := 	TRUE;

Control.b_DCFancoilEnable 		:= TRUE;
Control.b_DCPumpEnable 			:= TRUE;
END_ACTION

ACTION ECM_RequestPower:
SFCActive:= True;
IPSDemand.b_Demand_24V := TRUE;
END_ACTION

ACTION ECM_Shutdown:
Control.b_CloseBatteryLoopValve 	:= 	FALSE;
Control.b_CloseFancoilLoopValve 	:= 	FALSE;
Control.b_CloseInverterLoopValve := 	FALSE;

Control.b_DCFancoilEnable 		:= 	FALSE;
Control.b_DCPumpEnable 			:= 	FALSE;

IPSDemand.b_Demand_24V 		:= 	FALSE;
SFCActive:= False;
END_ACTION

METHOD SFCEnable : BOOL
VAR_INPUT
	Enable	:	Bool;
END_VAR
IF Enable THEN
	SFCInit := FALSE;
ELSE
	SFCActive:= FALSE;
	SFCInit := TRUE;
END_IF
END_METHOD

END_FUNCTION_BLOCK

// ---- POUs/Objects/CoolingSystem/SFC/FB_PowerModeConditioningSFC.TcPOU
FUNCTION_BLOCK FB_PowerModeConditioningSFC
VAR_IN_OUT
	//IPSState						:	ST_InternalPowerStatus;
	IPSDemand						:	ST_PowerDemand;
	
	ConditioningRequirements		: 	ST_ConditioningRequirements;
	Control							:	ST_CoolingSystem_Control;
	Get								:	ST_CoolingSystemGet;	

END_VAR
VAR_OUTPUT
	SFCActive	:	BOOL;
END_VAR

VAR
	AverageSystemLoadData	:	ARRAY[0..240] OF LREAL;
	// Gemiddelde load over 60s, Koelsysteem is toch traag
	AverageSystemLoadParams : TC2_ControllerToolbox.ST_CTRL_MOVING_AVERAGE_PARAMS := (tCtrlCycleTime := TIME#250ms, tTaskCycleTime := TIME#250ms, nSamplesToFilter := 240, pWorkArray_ADR := ADR(AverageSystemLoadData), nWorkArray_SIZEOF := sizeof(AverageSystemLoadData));
	AverageSystemLoad: FB_CTRL_MOVING_AVERAGE;
	
	CorrectionPIDParams : TC2_ControllerToolbox.ST_CTRL_PID_PARAMS := (tCtrlCycleTime := CoolingSystemParams.PIDLoopTime, tTaskCycleTime := CoolingSystemParams.PIDLoopTime, fKp := CoolingSystemParams.PIDControlKfactor, tTn := CoolingSystemParams.PIDControlTn, tTv := CoolingSystemParams.PIDControlTv, tTd := CoolingSystemParams.PIDControlTd, fOutMaxLimit := CoolingSystemParams.PIDControlLimitMax, fOutMinLimit := CoolingSystemParams.PIDControlLimitMin);
	CorrectionPID: FB_CTRL_PID;
	//NewSetpoint: REAL;
	
	r_ExpectedBaseCoolantTemp	:	REAL;
	
	b_ValveStateOK	:	Bool;
END_VAR

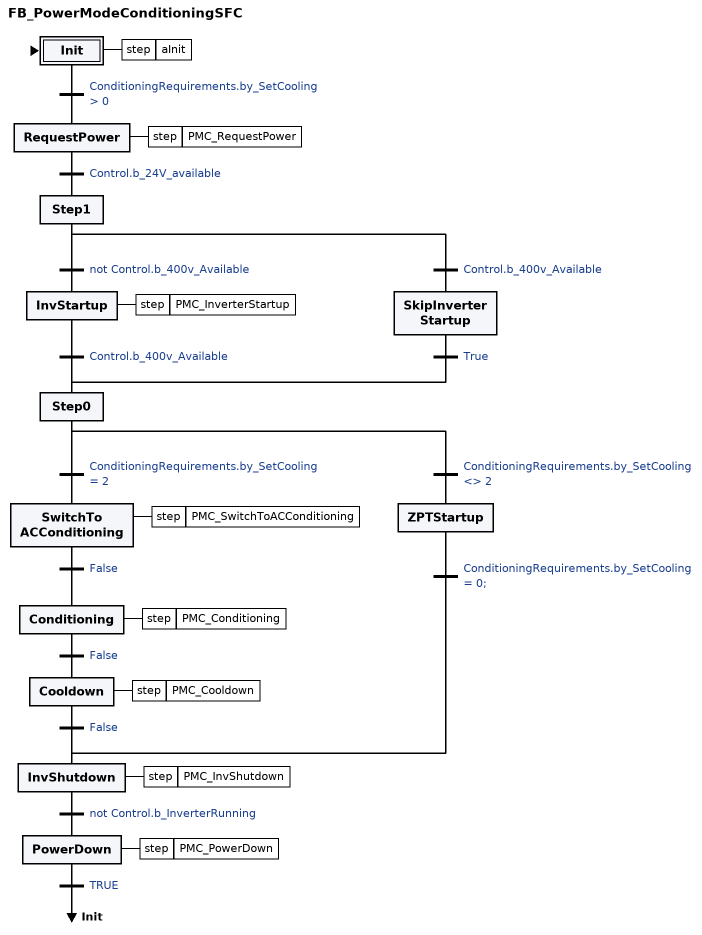
INITIAL_STEP Init:
    aInit(N);  // step action
END_STEP
TRANSITION FROM Init TO RequestPower
    := ConditioningRequirements.by_SetCooling > 0;
END_TRANSITION
STEP RequestPower:
    PMC_RequestPower(N);  // step action
END_STEP
TRANSITION FROM RequestPower TO Step1
    := Control.b_24V_available;
END_TRANSITION
STEP Step1:
END_STEP
TRANSITION FROM Step1 TO InvStartup
    := not Control.b_400v_Available;
END_TRANSITION
STEP InvStartup:
    PMC_InverterStartup(N);  // step action
END_STEP
TRANSITION FROM InvStartup TO Step0
    := Control.b_400v_Available;
END_TRANSITION
TRANSITION FROM Step1 TO SkipInverterStartup
    := Control.b_400v_Available;
END_TRANSITION
STEP SkipInverterStartup:
END_STEP
TRANSITION FROM SkipInverterStartup TO Step0
    := True;
END_TRANSITION
STEP Step0:
END_STEP
TRANSITION FROM Step0 TO SwitchToACConditioning
    := ConditioningRequirements.by_SetCooling = 2;
END_TRANSITION
STEP SwitchToACConditioning:
    PMC_SwitchToACConditioning(N);  // step action
END_STEP
TRANSITION FROM SwitchToACConditioning TO Conditioning
    := False;
END_TRANSITION
STEP Conditioning:
    PMC_Conditioning(N);  // step action
END_STEP
TRANSITION FROM Conditioning TO Cooldown
    := False;
END_TRANSITION
STEP Cooldown:
    PMC_Cooldown(N);  // step action
END_STEP
TRANSITION FROM Cooldown TO InvShutdown
    := False;
END_TRANSITION
TRANSITION FROM Step0 TO ZPTStartup
    := ConditioningRequirements.by_SetCooling <> 2;
END_TRANSITION
STEP ZPTStartup:
END_STEP
TRANSITION FROM ZPTStartup TO InvShutdown
    := ConditioningRequirements.by_SetCooling = 0;
END_TRANSITION
STEP InvShutdown:
    PMC_InvShutdown(N);  // step action
END_STEP
TRANSITION FROM InvShutdown TO PowerDown
    := not Control.b_InverterRunning;
END_TRANSITION
STEP PowerDown:
    PMC_PowerDown(N);  // step action
END_STEP
TRANSITION FROM PowerDown TO Init
    := TRUE;
END_TRANSITION
// branch label Branch0_PowerModeSFC

ACTION aInit:
SFCActive := False;
END_ACTION

ACTION PMC_Conditioning:


{warning "PowerModePID nog uitwerken en testen"}
{warning "placeholder voor de pid"}
// PID testen kan pas als het systeem helemaal draait. Voor nu geen tijd in stoppen maar testen met fixed setpoint.
//Gezien de modulerende regeling van de warmtepomp is een uitgebreide PID misschien amper nodig, enkel een long-term reactie op daadwerkelijke accutemperatuur.

Control.e_HeatpumpMode := eHeatpumpMode.Cooling;
Control.r_HeatPumpSetpoint := 10.0;

//initiate cooldown
IF ConditioningRequirements.by_SetCooling < 2 THEN
	ConditioningRequirements.by_PSCoolingPowerMode := 1;
	SFCTip := TRUE;
END_IF

//if coolantpressure drops below startup minimum, start DC pump and shutdown system immediately!
IF Control.r_CoolantPressure < (CoolingSystemParams.StartupPumpMinimumPressure + Control.r_CoolantIdlePressure) THEN
	control.b_DCPumpEnable := TRUE;
	get.Events.b_InverterCoolingLoopError := TRUE;
	ConditioningRequirements.by_PSCoolingPowerMode := 0;
END_IF


//PID disabled for now. Test with fixed setpoint first.


//AverageSystemLoad(stParams := AverageSystemLoadParams, fIn := Control.r_OutputPowerLevel);
//r_ExpectedBaseCoolantTemp := LREAL_TO_REAL(CoolingSystemParams.BattGoalTemp-(AverageSystemLoad.fOut /100 * CoolingSystemParams.CoolantFullPowerTemperatureOffset));

//Coolingsystem dictated by battery
//CorrectionPID.stParams := CorrectionPIDParams;
//CorrectionPID.fSetpointValue := CoolingSystemParams.BattGoalTemp;
//CorrectionPID.fActualValue := BattAvgTemp;

//CorrectionPID.stParams.fKp := CoolingSystemParams.PIDControlKfactor;

//CorrectionPID.stParams.tCtrlCycleTime := CoolingSystemParams.PIDLoopTime;
//CorrectionPID.stParams.tTn := CoolingSystemParams.PIDControlTn;//Integral coefficient
//CorrectionPID.stParams.tTv := CoolingSystemParams.PIDControlTv;//Derivative coefficient 
//CorrectionPID.stParams.tTd := CoolingSystemParams.PIDControlTd;//Damping time 
//CorrectionPID.stParams.fOutMaxLimit := CoolingSystemParams.PIDControlLimitMax;      //max correctie
//CorrectionPID.stParams.fOutMinLimit := CoolingSystemParams.PIDControlLimitMin;     // min correctie 
//CorrectionPID.stParams.bDInTheFeedbackPath := FALSE; //voorkomt oscillatie bij setpoint wijziging door dif loop. maar die is hier niet in gebruik.
//CorrectionPID.stParams.bPInTheFeedbackPath := FALSE; //?


//CorrectionPID(	stParams := CorrectionPIDParams, 
//				fSetpointValue := CoolingSystemParams.BattGoalTemp, 
//				fActualValue := Control.r_BMSBatteryTemperature);
				

//Control.r_HeatPumpSetpoint := r_ExpectedBaseCoolantTemp - CorrectionPID.fOut;
END_ACTION

ACTION PMC_Cooldown:

//first setup. Basic setpoint to return to idle temperatures
// After battery is done, enclosure is checked as well. May not be neccessary.
//Inverter is currently not checked, may be desirable after long runs.

IF ConditioningRequirements.Battery = eConditioningRequirement.Cooling THEN
	Control.b_CloseBatteryLoopValve := FALSE;
	Control.e_HeatpumpMode := eHeatpumpmode.Cooling;
	Control.r_HeatPumpSetpoint := 10.0;
ELSIF ConditioningRequirements.Battery = eConditioningRequirement.Heating THEN
	Control.b_CloseBatteryLoopValve := FALSE;
	Control.e_HeatpumpMode := eHeatpumpmode.Heating;
	Control.r_HeatPumpSetpoint := 35.0;
ELSE
	//battery conditioning done, close valve to speed up other conditioning loops
	Control.b_CloseBatteryLoopValve := TRUE;
	IF ConditioningRequirements.Enclosure = eConditioningRequirement.Heating THEN
		Control.e_HeatpumpMode := eHeatpumpmode.Heating;
		Control.r_HeatPumpSetpoint := 35.0;
	ELSIF ConditioningRequirements.Enclosure = eConditioningRequirement.Cooling THEN
		Control.e_HeatpumpMode := eHeatpumpmode.Cooling;
		Control.r_HeatPumpSetpoint := 10.0;
	ELSE
		//if enclosure and battery are ok. Inverter is presumably already cooled down enough. 
		Control.e_HeatpumpMode := eHeatpumpmode.standby;
		SFCTip := TRUE;	

	{warning "Add inverter temp check?"};
	//If not, keep running in current mode for longer
	//	IF PSGet.r_TemperatureMax < CoolingSystemParams.InverterIdleShutdownTemp THEN
		//	ConditioningModeRequired := eConditioningStates.OFF;
		//END_IF
	END_IF	
END_IF
END_ACTION

ACTION PMC_InverterStartup:
Control.b_CloseBatteryLoopValve 	:= TRUE;
Control.b_CloseFancoilLoopValve 	:= TRUE;
Control.b_CloseInverterLoopValve 	:= FALSE;

Control.b_DCFancoilEnable := FALSE;
//Control.b_ACFancoilEnable := FALSE;

Control.b_DCPumpEnable := TRUE;
Control.b_ACPumpEnable := FALSE;


Control.b_HeatPumpPowerEnable := FALSE;

//if both are ok, the inverter should have enough flow to start
IF Control.r_CoolantPressure > (CoolingSystemParams.StartupPumpMinimumPressure + Control.r_CoolantIdlePressure) AND Control.b_InverterLoopEnabled THEN
	//Inverter may commence modulating, but no power delivery yet.
	ConditioningRequirements.by_PSCoolingPowerMode := 1;
END_IF
END_ACTION

ACTION PMC_InvShutdown:
Control.b_CloseBatteryLoopValve := TRUE;
Control.b_CloseFancoilLoopValve := TRUE;
Control.b_CloseBatteryLoopValve := FALSE;

Control.b_DCFancoilEnable := FALSE;
//Control.b_ACFancoilEnable := FALSE;

Control.b_DCPumpEnable := TRUE;
Control.b_ACPumpEnable := FALSE;

Control.b_HeatPumpPowerEnable := FALSE;
Control.e_HeatpumpMode := eHeatpumpmode.standby;

//Inverter may shutdown now
ConditioningRequirements.by_PSCoolingPowerMode := 0;
END_ACTION

ACTION PMC_PowerDown:

Control.b_CloseBatteryLoopValve 	:= FALSE;
Control.b_CloseFancoilLoopValve 	:= FALSE;
Control.b_CloseBatteryLoopValve 	:= FALSE;

Control.b_DCFancoilEnable 		:= FALSE;
//Control.b_ACFancoilEnable		:= FALSE;

Control.b_DCPumpEnable 			:= FALSE;
Control.b_ACPumpEnable 			:= FALSE;

Control.b_HeatPumpPowerEnable	:= FALSE;


IPSDemand.b_Demand_24V 			:= FALSE;

SFCActive := FALSE;
END_ACTION

ACTION PMC_RequestPower:
SFCActive := TRUE;
IPSDemand.b_Demand_24V := TRUE;
IPSDemand.b_Demand_400V := TRUE;
END_ACTION

ACTION PMC_SwitchToACConditioning:





//First enable both pumps to see if AC pump works (by checking pressure increase)
Control.b_ACPumpEnable 			:= TRUE;
Control.b_DCPumpEnable 			:= TRUE;

IF Control.r_CoolantPressure > (CoolingSystemParams.MainPumpMinimumPressure + Control.r_CoolantIdlePressure) THEN
	Control.b_CloseBatteryLoopValve 	:= FALSE;
	Control.b_CloseFancoilLoopValve 	:= FALSE;
	Control.b_CloseInverterLoopValve 	:= FALSE;
		
	Control.b_HeatPumpPowerEnable 	:= TRUE;
	Control.e_HeatpumpMode := eHeatpumpmode.standby;
	
	Control.b_DCPumpEnable 			:= FALSE;
	
	Control.b_DCFancoilEnable 		:= TRUE;

	//if all loops are enabled, system is ready for operation
	IF Control.b_BatteryLoopEnabled AND Control.b_InverterLoopEnabled AND Control.b_FancoilLoopEnabled THEN;
		ConditioningRequirements.by_PSCoolingPowerMode := 2;
		SFCTip := TRUE;
	END_IF
END_IF
END_ACTION

METHOD SFCEnable : BOOL
VAR_INPUT
	Enable	:	Bool;
END_VAR
IF Enable THEN
	SFCInit := FALSE;
ELSE
	SFCActive:= FALSE;
	SFCInit := TRUE;
END_IF
END_METHOD

END_FUNCTION_BLOCK

// ---- POUs/Objects/CoolingSystem/FB_CoolingSystem_IO.TcPOU
FUNCTION_BLOCK FB_CoolingSystem_IO
VAR
	Inputs							AT %I*	:	ST_CoolingSystemInputs;
	Outputs							AT %Q* 	:	ST_CoolingSystemOutputs;
	ControlData: INT;
	ScalePressure: FB_CTRL_SCALE;
	PressureScaleParams: ST_CTRL_SCALE_PARAMS := (tTaskCycleTime := TIME#1ms, tCtrlCycleTime := TIME#1ms, fInMin := 0, fInMax := 4095, fOutMin := 0, fOutMax := 10);
	ScaleTemp: FB_CTRL_SCALE;
	TempScaleParams: ST_CTRL_SCALE_PARAMS;
	

	BattValveDelayTimer: TP := (PT := CoolingSystemParams.MaximumValveOperatingTime);
	FancoilValveDelayTimer: TP := (PT := CoolingSystemParams.MaximumValveOperatingTime);
	InvValveDelayTimer: TP := (PT := CoolingSystemParams.MaximumValveOperatingTime);
END_VAR

VAR_IN_OUT
	IO			:	ST_CoolingSystem_Control;
	Events		: 	ST_CoolingSystemEvents; 
END_VAR
VAR
	IdlePressureMeasurementDelay: ST_CoolingSystemEvents;
END_VAR



//Convert and scale pressure sensor data
{warning "TODO: FB_CTRLSCALE werkt nog niet"}
IO.r_CoolantPressure := (INT_TO_REAL(Inputs.CoolingLoopPressureSensor)/409.6);
//ScalePressure(fIn := Inputs.CoolingLoopPressureSensor, stParams:= PressureScaleParams, fOut=>IO.r_CoolantPressure);

IF (NOT IO.b_ACPumpEnable) AND (NOT IO.b_DCPumpEnable) THEN
	IO.r_CoolantIdlePressure := IO.r_CoolantPressure;
END_IF

//Cooling system pressure check. Lowest pressure will occur with pumps off.
//if this dips below the minimum pressure, the system has lost coolant and should be fixed.
Events.b_CoolingLoopIdlePressureWarning := (IO.r_CoolantPressure < CoolingSystemParams.MinimumSystemBasePressureWarningLevel);
Events.b_CoolingLoopIdlePressureError 	:= (IO.r_CoolantPressure < CoolingSystemParams.MinimumSystemBasePressureErrorLevel);

//Convert and scale coolant tank temperature data
{warning "TODO: FB_CTRLSCALE werkt nog niet"}
IO.r_CoolantTemperature := (INT_TO_REAL(Inputs.CoolingLoopTemperatureSensor)/40.96)-40;
//ScalePressure(fIn := Inputs.CoolingLoopTemperatureSensor, stParams:= TempScaleParams, fOut=>IO.r_CoolantTemperature);

//Pump control
Outputs.ACPumpEnable := IO.b_ACPumpEnable;
Outputs.DCPumpEnable := IO.b_DCPumpEnable;

//FanControl
Outputs.DCFanEnable := IO.b_DCFancoilEnable;


//Battloop valve control
//First set output and edge detectors. The edge detectors trigger a grace period in which the valve state is allowed to diverge from requested state
Outputs.BattLoopValveClose := IO.b_CloseBatteryLoopValve;

//Feedback is inverse from output. If they stay the same for too long --> Valve is stuck or inoperative
IO.b_BatteryLoopEnabled := Inputs.BattLoopValveFB;
BattValveDelayTimer(IN := IO.b_CloseBatteryLoopValve = Inputs.BattLoopValveFB);
Events.b_BattLoopValveStuck := BattValveDelayTimer.Q;


//Inverter loop valve control
//First set output and edge detectors. The edge detectors trigger a grace period in which the valve state is allowed to diverge from requested state
Outputs.InvLoopValveClose := IO.b_CloseInverterLoopValve;

//Feedback is inverse from output. If they stay the same for too long --> Valve is stuck or inoperative
IO.b_InverterLoopEnabled := Inputs.InvLoopValveFB;
InvValveDelayTimer(IN := IO.b_CloseInverterLoopValve = Inputs.InvLoopValveFB);
Events.b_InverterLoopValveStuck := InvValveDelayTimer.Q;


//Fancoil loop valve control
//First set output and edge detectors. The edge detectors trigger a grace period in which the valve state is allowed to diverge from requested state
Outputs.FancoilLoopValveClose := IO.b_CloseFancoilLoopValve;

//Feedback is inverse from output. If they stay the same for too long --> Valve is stuck or inoperative
IO.b_FancoilLoopEnabled := Inputs.FancoilLoopValveFB;
FancoilValveDelayTimer(IN := IO.b_CloseFancoilLoopValve = Inputs.FancoilLoopValveFB);
Events.b_FancoilLoopValveStuck := FancoilValveDelayTimer.Q;




//400V fuse feedback
Events.b_CoolingSystemFuseFailure := NOT Inputs.CoolingSystem400VFuseFB;

END_FUNCTION_BLOCK

// ---- POUs/Objects/ExternalControl/FB_ExternalControl.TcPOU
FUNCTION_BLOCK FB_ExternalControl
VAR

END_VAR
VAR
END_VAR

END_FUNCTION_BLOCK

// ---- POUs/Objects/InternalPowerSupply/FB_InternalPowerSupply.TcPOU
FUNCTION_BLOCK FB_InternalPowerSupply
VAR CONSTANT
	//w_ID														: WORD := eObject_ID.InternalPowerSupply;
END_VAR

VAR
	IO: FB_InternalPowerSupply_IO;
	InternalPowerDemand: ST_PowerDemand;
	b_EMStopActive : BOOL := FALSE;
END_VAR

VAR_INPUT
	Set					:	ST_InternalPowerSupply_Set;
	BMSPowerstate		:	eHVDC_Powerstatus;
	b_ConditioningOnBatteryAllowed:	BOOL;
END_VAR

VAR_OUTPUT
	Get					:	ST_InternalPowerSupply_Get;
	b_HVDC_Enable		:	BOOL;
END_VAR

VAR
	ShutdownRequested	: BOOL := FALSE;	
	UPS					: FB_UPS;
END_VAR

(*
FB_InternalPowersupply
	Inputs:
		Power demand set by each applicable block, each with 3 booleans for 24V, 400VAc and HVDC:
			CoolingSystemPowerDemand	:	st_PowerDemand;
			PowerStackPowerDemand		:	st_PowerDemand;	
			UPSPowerDemand				:	st_PowerDemand;
			InternalPowerDemand			:	st_PowerDemand;
		
		Main system settings:	
			b_GeneralPowerEnable			: 	BOOL;	No power allowed without this being true. UPS only mode
		
		Input from powerstack. 400VAC available on busbar (via inverter or grid supply)	
			b_InternalBusbarACAvailable
		
		b_ShutdownUPS
			Kills UPS power, but only if other supplies are already down. 
	
	Outputs
		b_24VdcAvailable		
		b_HVDCAvailable			
		b_400VACAvailable		
			
		b_BMSForceOff 			//Output to FB_BMS to kill BMS supply voltage.
	
		UPS			//UPS data structure
	
		Events		
*)

//only if other power supplies are already down, UPS disable is allowed. Unwanted on live system.
IF (NOT (get.b_24VdcAvailable OR get.b_400VACAvailable OR get.b_HVDCAvailable)) AND set.b_ShutdownUPS THEN
	UPS.Shutdown();
END_IF

UPS(b_24v_available := get.b_24VdcAvailable, Get => get.UPS);
IO();
ACPowerControl();
DCPowerControl();
HVDCPowerControl();

METHOD PRIVATE ACPowerControl : BOOL
VAR
	AC_StartupDelay: TON := (PT := IPSParams.ACStartupDelay);
END_VAR
//AC control function
//Initial Diagnostics by reading fuse feedback
get.Events.b_GridInputFuseTripped 	:= NOT IO.GridFuseOK;
get.Events.b_CEEInputFuseTripped 	:= NOT IO.CeeFuseOK;

IF set.b_GeneralPowerEnable OR b_EMStopActive THEN
	//Grid power has priority over CEE plug
	IF 	IO.GridFuseOK AND set.b_InternalBusbarACAvailable THEN
		IO.SetACConnectionMode := 1;	//switch to grid AC
		AC_StartupDelay.IN := TRUE;	
	ELSIF IO.CEE_ACAvailable THEN 
		IO.SetACConnectionMode := 2;	//switch to CEE AC
		
		//not anymore
		//IF NOT Config.b_NeutralTransformer THEN //internal neutral transformer has longer startup time
		//	AC_StartupDelay.PT := IpsParams.ACStartupDelay+IPSParams.IntZPTStartupDelay;	
		//END_IF
		
		AC_StartupDelay.IN := TRUE;
	ELSE
		IO.SetACConnectionMode := 0;	//disable
		AC_StartupDelay.IN := FALSE;
	END_IF
ELSE 
	IO.SetACConnectionMode := 0;	//disable
	AC_StartupDelay.IN := FALSE;
END_IF

//after startup delay, internal 400VAC is available
get.b_400VACAvailable := AC_StartupDelay.Q;
END_METHOD

METHOD DCPowerControl : BOOL
VAR_INPUT
END_VAR
VAR
	DC_Required: BOOL;
	DCPSU_StartupDelay: TON := (PT := IPSParams.DCPSU_StartupDelay);
	ACPSU_StartupDelay: TON := (PT := IPSParams.ACPSU_StartupDelay);
END_VAR
ACPSU_StartupDelay.IN := get.b_400VACAvailable;
DCPSU_StartupDelay.IN := get.b_HVDCAvailable;

//if psu is not online after the startup delay, raise the fault status.
get.Events.b_ACPSUFault := ACPSU_StartupDelay.Q AND NOT IO.ACPSU_OK;
get.Events.b_DCPSUFault := DCPSU_StartupDelay.Q AND NOT IO.DCPSU_OK;

//if any of the psu's is online, 24V is available
get.b_24VdcAvailable := IO.ACPSU_OK OR IO.DCPSU_OK;

//All parts can demand 24V
DC_Required :=	set.CoolingSystemPowerDemand.b_Demand_24V OR 
				set.PowerStackPowerDemand.b_Demand_24V OR 
				set.UPSPowerDemand.b_Demand_24V;

//if no 400VAC available during 24VDC request, request HVDC ON for LVDC power				
internalPowerDemand.b_Demand_HVDC := DC_Required AND NOT get.b_400VACAvailable;
END_METHOD

METHOD PUBLIC EMstop : BOOL
VAR_INPUT
END_VAR
//return true if done
b_EMStopActive := TRUE;

//return true when all supplies are lost.
EMStop := not(get.b_24VdcAvailable OR get.b_400VACAvailable OR get.b_HVDCAvailable);
END_METHOD

METHOD GetDiagnostics 
VAR_IN_OUT
	AddError		: ARRAY [*] OF FB_AddErrorST;
	a_ActiveEvents	: ARRAY [*] OF ST_ErrorStruct;
	w_Index			: WORD;
END_VAR

VAR_OUTPUT
	b_errorActive	: BOOL;
	b_warningActive	: BOOL;
END_VAR

VAR
	by_errCt	: BYTE;
	by_warnCt	: BYTE;
	w_ID		: WORD;
END_VAR

//check if this call works:
UPS.GetDiagnostics(AddError := AddError, a_ActiveEvents := a_ActiveEvents, w_Index := w_Index, b_errorActive => b_errorActive, b_warningActive => b_warningActive);

(*IPS*)
	(*AC PSU fault*)		AddError[w_Index](
			in_b_ErrorTrig			:= Get.Events.b_ACPSUFault,
			out_ST_Error			:= a_ActiveEvents[w_Index],
			w_ID					:= 1 + w_ID,
			s_Message				:= 'AC PSU fault',
			e_sev					:= eSeverity.Warning,
			);
		IF AddError[w_Index].b_out THEN by_WarnCt := by_WarnCt + 1; END_IF;
		w_Index := w_Index +1;
		
	(*DC PSU fault*)		AddError[w_Index](
			in_b_ErrorTrig			:= Get.Events.b_DCPSUFault,
			out_ST_Error			:= a_ActiveEvents[w_Index],
			w_ID					:= 1 + w_ID,
			s_Message				:= 'DC PSU fault',
			e_sev					:= eSeverity.Warning,
			);
		IF AddError[w_Index].b_out THEN by_WarnCt := by_WarnCt + 1; END_IF;
		w_Index := w_Index +1;
	
	(*24V fault*)		AddError[w_Index](
			in_b_ErrorTrig			:= Get.Events.b_DCPSUFault AND Get.Events.b_ACPSUFault,
			out_ST_Error			:= a_ActiveEvents[w_Index],
			w_ID					:= 1 + w_ID,
			s_Message				:= '24V supply failed',
			e_sev					:= eSeverity.QuickShutdown,
			);
		IF AddError[w_Index].b_out THEN by_errCt := by_errCt + 1; END_IF;
		w_Index := w_Index +1;	
		
	(*CEE fuse tripped*)		AddError[w_Index](
			in_b_ErrorTrig			:= Get.Events.b_CEEInputFuseTripped,
			out_ST_Error			:= a_ActiveEvents[w_Index],
			w_ID					:= 1 + w_ID,
			s_Message				:= 'CEE Standby power input fuse error',
			e_sev					:= eSeverity.Warning,
			in_b_AutoClear			:= TRUE,
			
			);
		IF AddError[w_Index].b_out THEN by_WarnCt := by_WarnCt + 1; END_IF;
		w_Index := w_Index +1;
	
	(*internal grid fuse fault*)		AddError[w_Index](
			in_b_ErrorTrig		:= Get.Events.b_GridInputFuseTripped,
			out_ST_Error			:= a_ActiveEvents[w_Index],
			w_ID					:= 1 + w_ID,
			s_Message				:= 'Internal supply Grid fuse error',
			e_sev					:= eSeverity.QuickShutdown,
			in_b_AutoClear			:= TRUE,
			);
		IF AddError[w_Index].b_out THEN by_errCt := by_errCt + 1; END_IF;
		w_Index := w_Index +1;
		
	(*EMSTOP HVDC shutdown failed*)		AddError[w_Index](
			in_b_ErrorTrig			:= Get.Events.b_HVDCShutdownTimeExceeded,
			out_ST_Error			:= a_ActiveEvents[w_Index],
			w_ID					:= 1 + w_ID,
			s_Message				:= 'HVDC shutdown sequence failed',
			e_sev					:= eSeverity.QuickShutdown,			//<-- already in emstop, but this is a severe error
			);
		IF AddError[w_Index].b_out THEN by_errCt := by_errCt + 1; END_IF;
		w_Index := w_Index +1;
END_METHOD

METHOD PRIVATE HVDCPowerControl : BOOL
VAR_INPUT
END_VAR

//The powerstack demands HVDC directly. 
IF b_EMStopActive THEN
	b_HVDC_Enable := FALSE;
ELSE
	b_HVDC_Enable := set.PowerStackPowerDemand.b_Demand_HVDC 
		OR (InternalPowerDemand.b_Demand_HVDC AND b_ConditioningOnBatteryAllowed AND NOT ShutdownRequested);
END_IF						

IF BMSPowerState = eHVDC_Powerstatus.ON THEN
	get.b_HVDCAvailable := TRUE;
ELSE
	get.b_HVDCAvailable := FALSE;
END_IF
END_METHOD

METHOD Reset : BOOL
VAR_INPUT
END_VAR
//reset system
//return true if ok

b_EMStopActive 					:= 	FALSE;
IO.b_InternalHVDCConnected		:=	TRUE;

Reset := NOT get.Events.b_GridInputFuseTripped;
END_METHOD

METHOD SystemShutdown : BOOL
VAR_INPUT
	b_force		:	Bool;
END_VAR

IF B_force THEN
	IO.SetACConnectionMode 		:= 	0;
	IO.b_InternalHVDCConnected	:=	FALSE;
	IO.Write();

	UPS.Shutdown();
ELSE
	//no unforced shutdown allowed if HVDC is still online.
	//if HVDC offline, disable AC inputs and decouple HV contactors
	//Wait for 400VAC and 24V to be offline, then kill the UPS
	IF NOT get.b_HVDCAvailable THEN
		IO.b_InternalHVDCConnected := 0;
		IO.SetACConnectionMode 		:= 	0;
		IF NOT get.b_400VACAvailable AND get.b_24VdcAvailable THEN
			UPS.Shutdown();
		END_IF
	END_IF
END_IF
END_METHOD

END_FUNCTION_BLOCK

// ---- POUs/Objects/InternalPowerSupply/FB_InternalPowerSupply_IO.TcPOU
FUNCTION_BLOCK FB_InternalPowerSupply_IO
VAR
	b_Write					AT %Q* : ARRAY[1..3] OF BOOL;	
	b_Read					AT %I* : ARRAY[1..5] OF BOOL;
END_VAR

VAR_INPUT
	// 0: No AC, 1: Grid AC, 2: CEE AC
	SetACConnectionMode: BYTE := 0;
	b_InternalHVDCConnected : BOOL := FALSE;
END_VAR

VAR_OUTPUT
	DCPSU_OK: BOOL;
	ACPSU_OK: BOOL;
	GridFuseOK: BOOL;
	CeeFuseOK: BOOL;
	CEE_ACAvailable: BOOL;
END_VAR

read();
write();

METHOD PRIVATE Read : BOOL
DCPSU_OK := b_read[1];
ACPSU_OK := b_read[2];
GridFuseOK := b_read[3];
CeeFuseOK := b_read[4];
CEE_ACAvailable := b_read[5];
END_METHOD

METHOD Write : BOOL
VAR_INPUT
END_VAR
//B_write[1] = Main supply enable (53Q2)
//B_write[2] = CEE supply enable (53Q1)

CASE SetACConnectionMode OF
	0: b_Write[2] := FALSE; b_Write[1] := FALSE;
	1: b_Write[2] := FALSE; b_Write[1] := TRUE;
	2: b_Write[2] := TRUE; 	b_Write[1] := FALSE;
END_CASE

//HVDC disconnect contactors, Only opened in emergency situations when HVDC disconnect fails.
//Opening these contactors also removes insulation monitor functionality.
b_Write[3] := b_InternalHVDCConnected;
END_METHOD

END_FUNCTION_BLOCK

// ---- POUs/Objects/InternalPowerSupply/UPS/FB_UPS.TcPOU
FUNCTION_BLOCK FB_UPS
VAR_INPUT
	b_24V_Available	:	BOOL;
END_VAR
VAR_OUTPUT
	Get	: ST_UPSGET;
END_VAR
VAR
	DisableUPS		AT %Q* : BOOL;
	UPSData			AT %I* : ST_UPSDATA;	
	InputTimer		: TON := (PT := TIME#100ms);
END_VAR

//no need to call this FB from the main sequence
//This FB is controlled via the internal power supply

Get.r_BatteryVoltage 	:= 	UPSData.ui_BatteryVoltage;
Get.r_InputVoltage		:=	UPSData.ui_InputVoltage;
Get.r_OutputVoltage		:=	UPSData.ui_OutputVoltage;
Get.ui_SOC 				:= GetSOC();


//if r_SOC below threshold, battery is critically low. System should shutdown.
IF Get.ui_SOC  < IPSParams.usi_UPSBattLowErrorSOC THEN
	get.Events.b_BatteryLowError := TRUE;
END_IF

//if r_SOC below threshold, charging request was denied. System is draining. Consider shutdown.
IF Get.ui_SOC  < IPSParams.usi_UPSBattLowwarningSOC THEN
	get.Events.b_BatteryLowWarning := TRUE;
END_IF

//if r_SOC below threshold, request charging power from IPS
IF Get.ui_SOC  < IPSParams.usi_UPSBattLowinfoSOC THEN
	get.UPSPowerDemand.b_Demand_24V := TRUE;
	get.Events.b_BatteryLowNotice := TRUE;
//if r_SOC above threshold remove charging request to prevent prolonged HVDC usage.
ELSIF Get.ui_SOC  > IPSParams.usi_UPSBattOKSOC THEN
	get.UPSPowerDemand.b_Demand_24V := FALSE;
	get.Events.b_BatteryLowNotice := FALSE;
END_IF

//if system is charging, disable low battery error. Wait for sufficient r_SOC before disabling the low battery warning
IF UPSData.udi_StatusFunctions.5 THEN 
	get.Events.b_BatteryLowError := FALSE;
END_IF

IF get.r_BatteryVoltage < 16 THEN
	get.Events.b_NoBatteryError := TRUE;
ELSE 
	get.Events.b_NoBatteryError := FALSE;
END_IF

//UPS input voltage should be OK shortly after IPS 24V coming online. Otherwise there is a problem
InputTimer(in:= b_24V_Available);
get.Events.b_InputVoltageError := InputTimer.Q AND (UPSData.ui_InputVoltage < 20);

METHOD GetDiagnostics 
VAR_IN_OUT
	AddError		: ARRAY [*] OF FB_AddErrorST;
	a_ActiveEvents	: ARRAY [*] OF ST_ErrorStruct;
	w_Index			: WORD;
END_VAR

VAR_OUTPUT
	b_errorActive	: BOOL;
	b_warningActive	: BOOL;
END_VAR

VAR
	by_errCt	: BYTE;
	by_warnCt	: BYTE;
	w_ID		: WORD;
END_VAR
(*UPS*)
	(*Low battery error*)		AddError[w_Index](
			in_b_ErrorTrig			:= Get.Events.b_BatteryLowError,
			out_ST_Error			:= a_ActiveEvents[w_Index],
			w_ID					:= 1 + w_ID,
			s_Message				:= 'UPS Low battery error',
			e_sev					:= eSeverity.Warning,	//<-- not really applicable
			in_b_AutoClear			:= TRUE,
			);
		IF AddError[w_Index].b_out THEN by_WarnCt := by_WarnCt + 1; END_IF;
		w_Index := w_Index +1;
		
	(*low battery warning*)		AddError[w_Index](
			in_b_ErrorTrig			:= Get.Events.b_BatteryLowWarning,
			out_ST_Error			:= a_ActiveEvents[w_Index],
			w_ID					:= 2 + w_ID,
			s_Message				:= 'UPS Low battery warning',
			e_sev					:= eSeverity.Info,
			in_b_AutoClear			:= TRUE,
			);
		w_Index := w_Index +1;
	
	(*UPS input undervoltage*)		AddError[w_Index](
			in_b_ErrorTrig			:= Get.Events.b_InputVoltageError,
			out_ST_Error			:= a_ActiveEvents[w_Index],
			w_ID					:= 3 + w_ID,
			s_Message				:= 'UPS input undervoltage error',
			e_sev					:= eSeverity.Warning,
			in_b_AutoClear			:= TRUE,
			);
		IF AddError[w_Index].b_out THEN by_WarnCt := by_WarnCt + 1; END_IF;
		w_Index := w_Index +1;
	
	(*no UPS battery*)		AddError[w_Index](
			in_b_ErrorTrig		:= Get.Events.b_NoBatteryError,
			out_ST_Error			:= a_ActiveEvents[w_Index],
			w_ID					:= 4 + w_ID,
			s_Message				:= 'UPS no battery error',
			e_sev					:= eSeverity.Warning,
			);
		IF AddError[w_Index].b_out THEN by_WarnCt := by_WarnCt + 1; END_IF;
		w_Index := w_Index +1;
END_METHOD

METHOD GetSoC : USINT
VAR

END_VAR

//basic lineaire r_SOC berekening voor nu
IF UPSData.udi_StatusFunctions.5 THEN
	//charging
	//26V is 100%
	//23V is 0%
	GetSoC := REAL_TO_USINT((get.r_BatteryVoltage - 23)*33.3);
ELSE
	//discharging
	//25.7V is 100%
	//22.7V is 0%
	GetSoC := REAL_TO_USINT((get.r_BatteryVoltage - 22.7)*33.3);
END_IF
END_METHOD

METHOD Shutdown : BOOL

DisableUPS := True;
END_METHOD

END_FUNCTION_BLOCK

// ---- POUs/Objects/PowerQualityMonitor/FB_Beckhoff_EL3443_0010/FB_EL3443_0010.TcPOU
FUNCTION_BLOCK FB_EL3443_0010
VAR_INPUT
	b_enable	:	BOOL;
END_VAR

VAR
	EL3443FaultCounter			: UINT := 0;
END_VAR
VAR_OUTPUT
	PhaseStatus				AT %I* : ARRAY [1..3] OF ST_El3443_PhaseStatus;
	TotalStatus				AT %I* : ST_EL3443_TotalStatus;
	r_PhaseVoltage			AT %I* : ARRAY [1..3] OF REAL;
	r_LineVoltage			AT %I* : ARRAY [1..3] OF REAL;
	r_Current				AT %I* : ARRAY [1..4] OF REAL;
	r_ActivePower			AT %I* : ARRAY [1..3] OF REAL;
	r_ReactivePower			AT %I* : ARRAY [1..3] OF REAL;
	r_ApparentPower			AT %I* : ARRAY [1..3] OF REAL;
	r_PowerFactor			AT %I* : ARRAY [1..3] OF REAL;
	r_Frequency				AT %I* : REAL;
	r_ActiveEnergy			AT %I* : LINT;
	r_ActiveEnergyPositive 	AT %I* : LINT;
	r_ActiveEnergyNegative	AT %I* : LINT;
	ui_EL3443BoxState		AT %I* : UINT;
END_VAR

VAR_IN_OUT
	Get	: ST_PowerMonitor_get;
END_VAR


IF b_Enable THEN
	IF TotalStatus.bit_SystemState AND ui_EL3443BoxState = 16#8 THEN
		//Get Generator field voltage data from EL3443
		Get.InputField.r_PhaseVoltage[Phases.L1]:= r_PhaseVoltage[Phases.L1];
		Get.InputField.r_PhaseVoltage[Phases.L2]:=  r_PhaseVoltage[Phases.L2];
		Get.InputField.r_PhaseVoltage[Phases.L3]:=  r_PhaseVoltage[Phases.L3];
		Get.InputField.r_PhaseVoltage[Phases.AVG] := ( r_PhaseVoltage[Phases.L1] + r_PhaseVoltage[Phases.L2] +  r_PhaseVoltage[Phases.L3])/3;
		
		Get.InputField.r_LineVoltage[Phases.L1]:=  r_LineVoltage[Phases.L1];
		Get.InputField.r_LineVoltage[Phases.L2]:=  r_LineVoltage[Phases.L2];
		Get.InputField.r_LineVoltage[Phases.L3]:=  r_LineVoltage[Phases.L3];
		Get.InputField.r_LineVoltage[Phases.AVG] := ( r_LineVoltage[Phases.L1] +  r_LineVoltage[Phases.L2] +  r_LineVoltage[Phases.L3])/3;
		
		Get.InputField.r_Frequency :=  r_Frequency;
		
		Get.InputField.r_Current[Phases.L1]:= r_Current[Phases.L1];
		Get.InputField.r_Current[Phases.L2]:= r_Current[Phases.L2];
		Get.InputField.r_Current[Phases.L3]:= r_Current[Phases.L3];
		Get.InputField.r_Current[Phases.N]:= r_Current[Phases.N];	//<-- calculated N
		
		Get.InputField.r_ActivePhasePower[Phases.L1]:= r_ActivePower[Phases.L1];
		Get.InputField.r_ActivePhasePower[Phases.L2]:= r_ActivePower[Phases.L2];
		Get.InputField.r_ActivePhasePower[Phases.L3]:= r_ActivePower[Phases.L3];		
		Get.InputField.r_ActivePhasePower[Phases.AVG]:= (r_ActivePower[Phases.L1] + r_ActivePower[Phases.L2] + r_ActivePower[Phases.L3]);	
		Get.InputField.r_ActivePower := r_ActivePower[Phases.L1]+ r_ActivePower[Phases.L2] + r_ActivePower[Phases.L3];
		
